// TwinCAT 3 PLC project TcOpcUaServer_Testproject
// ProgramVersion: 3.1.4022.3
// libraries:
//   Tc2_MPBus, * (Beckhoff Automation GmbH)
//   Tc2_Standard, * (Beckhoff Automation GmbH)
//   Tc2_System, * (Beckhoff Automation GmbH)
//   Tc3_Interfaces, * (Beckhoff Automation GmbH)
//   Tc3_Module, * (Beckhoff Automation GmbH)
// project tree:
//   DUTs/Enums/ E_Enum_2.TcDUT, E_Operation.TcDUT, E_Enum_1.TcDUT (not stored)
//   DUTs/Structures/ ST_Complex_1.TcDUT, ST_Complex_3.TcDUT, ST_Complex_4.TcDUT, ST_Complex_5.TcDUT (not stored), ST_Complex_6.TcDUT, ST_Complex_7.TcDUT, ST_Complex_8.TcDUT, ST_MathematicResults.TcDUT (not stored), ST_MathOperation.TcDUT, ST_Complex_2.TcDUT (not stored)
//   GVLs/ GVL_alarm_condition.TcGVL (not stored), GVL_analog_items.TcGVL, GVL_historizing.TcGVL (not stored), GVL_inheritance.TcGVL (not stored), GVL_user_access.TcGVL, Settings.TcGVL (not stored), GVL_arrays.TcGVL, GVL_enums.TcGVL, GVL_methods.TcGVL (not stored), GVL_structures.TcGVL (not stored), GVL_nodes_dynamic.TcGVL, GVL_nodes_static.TcGVL
//   / PlcTask.TcTTO (not stored)
//   POUs/Inheritance/ FB_Base.TcPOU (not stored), FB_Derived.TcPOU (not stored)
//   POUs/ MAIN.TcPOU (not stored)
//   POUs/Methods/ FB_Mathematics.TcPOU (not stored), FB_Methods.TcPOU
//   POUs/Programs/ PRG_Dynamic.TcPOU, PRG_Static.TcPOU
// real-time tasks:
//   TASK PlcTask: cycle T#10ms, priority 20, ADS port 350

// ---- DUTs/Enums/E_Enum_2.TcDUT
TYPE E_Enum_2 :
(
	ZERO := 0,
	ONE := 1,
	TWO := 2,
	THREE := 3,
	THIRTEEN := 13,
	the_answer_to_life_the_universe_and_everything := 42
) INT;
END_TYPE

// ---- DUTs/Enums/E_Operation.TcDUT
TYPE E_Operation :
(
	Addition := 0,
	Substract,
	Multiply,
	Divide
);
END_TYPE

// ---- DUTs/Structures/ST_Complex_1.TcDUT
{attribute 'OPC.UA.DA' := '1'}
{attribute 'OPC.UA.DA.StructuredType' := '1'}
TYPE ST_Complex_1 :
STRUCT
	x 	: E_Enum_1;
	a 	: DINT;
	str : STRING;
	b 	: DINT;
END_STRUCT
END_TYPE

// ---- DUTs/Structures/ST_Complex_3.TcDUT
{attribute 'OPC.UA.DA' := '1'}
{attribute 'OPC.UA.DA.StructuredType' := '1'}
TYPE ST_Complex_3 :
STRUCT
	ErrorID : MP_ERROR;
END_STRUCT
END_TYPE

// ---- DUTs/Structures/ST_Complex_4.TcDUT
{attribute 'OPC.UA.DA' := '1'}
{attribute 'OPC.UA.DA.StructuredType' := '1'}
TYPE ST_Complex_4 :
STRUCT
	ErrorID : E_Enum_1;
END_STRUCT
END_TYPE

// ---- DUTs/Structures/ST_Complex_6.TcDUT
TYPE ST_Complex_6 :
STRUCT
	a : INT := 42;
	b : DINT := 43;
	c : REAL := 42.42;
	d : LREAL := 42.42;
	e : INT := 44;
	f : BOOL := TRUE;
END_STRUCT
END_TYPE

// ---- DUTs/Structures/ST_Complex_7.TcDUT
TYPE ST_Complex_7 :
STRUCT
	a : LREAL := 42.42;
	b : REAL := 42.42;
	c : REAL := 42.42;
END_STRUCT
END_TYPE

// ---- DUTs/Structures/ST_Complex_8.TcDUT
{attribute 'OPC.UA.DA' := '1'}
{attribute 'OPC.UA.DA.StructuredType' := '1'}
TYPE ST_Complex_8 :
STRUCT
	stComplex		: ST_Complex_1;
	strString5		: STRING[5]; (*String, max 5 chars*)
	eEnum	 		: E_Enum_1;
	strString3	 	: STRING[3]; (*String, max 3 chars*)
	arrComplex 		: ARRAY[0..1] OF ST_Complex_1;
	arrDint		 	: ARRAY[0..100] OF DINT;	
END_STRUCT
END_TYPE

// ---- DUTs/Structures/ST_MathOperation.TcDUT
{attribute 'OPC.UA.DA.Description' := 'Structure to describe a math operation having one operator and two oparands'}
TYPE ST_MathOperation :
STRUCT
	operator : E_OPERATION; (*define the operator for calculation*)
	a : LREAL; (*First operand*)
	b : LREAL; (*Second operand*)
END_STRUCT
END_TYPE

// ---- GVLs/GVL_analog_items.TcGVL
{attribute 'qualified_only'}
VAR_GLOBAL
	{attribute 'OPC.UA.DA' := '1'}
	{attribute 'OPC.UA.DA.AnalogItemType' := '1'}
	{attribute 'OPC.UA.DA.AnalogItemType.EngineeringUnits' := '20529'  }(*EngeneeringUnit = percent*)
	{attribute 'OPC.UA.DA.AnalogItemType.InstrumentRange' := '0:100'  }
	{attribute 'OPC.UA.DA.AnalogItemType.EURange' := '10:90'  }
	{attribute 'OPC.UA.DA.AnalogItemType.WriteBehavior' := '1'  } (*AnalogWrMode_AllowAny = 0,
																	AnalogWrMode_Clamp = 1,
																	AnalogWrMode_Reject = 2,*)
	{attribute 'OPC.UA.DA.Description' := 'Analog item type. Write mode is clamped to instrument range'}
	analog_percent : REAL := 50;
	
	{attribute 'OPC.UA.DA' := '1'}
	{attribute 'OPC.UA.DA.AnalogItemType' := '1'}
	{attribute 'OPC.UA.DA.AnalogItemType.EngineeringUnits' := '12851'  }(*EngeneeringUnit = gram_per_cubic_centimetre*)
	{attribute 'OPC.UA.DA.AnalogItemType.InstrumentRange' := '0:100'  }
	{attribute 'OPC.UA.DA.AnalogItemType.EURange' := '0:75'  }
	{attribute 'OPC.UA.DA.AnalogItemType.WriteBehavior' := '2'  } (*AnalogWrMode_AllowAny = 0,
																	AnalogWrMode_Clamp = 1,
																	AnalogWrMode_Reject = 2,*)
	{attribute 'OPC.UA.DA.Description' := 'Analog item type. Write is rejected when out of instrument range'}
	analog_gram_per_cubic_centimetre : REAL := 50;	
	
	{attribute 'OPC.UA.DA' := '1'}
	{attribute 'OPC.UA.DA.AnalogItemType' := '1'}
	{attribute 'OPC.UA.DA.AnalogItemType.EngineeringUnits' := '5257525'  }(*EngeneeringUnit = megabyte_per_second*)
	{attribute 'OPC.UA.DA.AnalogItemType.EURange' := '0:10'  }
	{attribute 'OPC.UA.DA.AnalogItemType.InstrumentRange' := '0:100'  }
	{attribute 'OPC.UA.DA.AnalogItemType.WriteBehavior' := '0'  } (*AnalogWrMode_AllowAny = 0,
																	AnalogWrMode_Clamp = 1,
																	AnalogWrMode_Reject = 2,*)
	{attribute 'OPC.UA.DA.Description' := 'Analog item type. Write mode allows writing out of Instrument range'}
	analog_mbps : REAL;	
	
	{attribute 'OPC.UA.DA' := '1'}
	{attribute 'OPC.UA.DA.AnalogItemType' := '1'}
	{attribute 'OPC.UA.DA.AnalogItemType.EngineeringUnits' := '20529'  }(*EngeneeringUnit = percent*)
	{attribute 'OPC.UA.DA.AnalogItemType.InstrumentRange' := '0:100'  }
	{attribute 'OPC.UA.DA.AnalogItemType.EURange' := '10:90'  }
	{attribute 'OPC.UA.DA.AnalogItemType.WriteBehavior' := '2'  } (*AnalogWrMode_AllowAny = 0,
																	AnalogWrMode_Clamp = 1,
																	AnalogWrMode_Reject = 2,*)
	{attribute 'OPC.UA.DA.Description' := 'Analog item of type Double. '}
	analog_dbl : LREAL := 50;	
	
	{attribute 'OPC.UA.DA' := '1'}
	{attribute 'OPC.UA.DA.AnalogItemType' := '1'}
	{attribute 'OPC.UA.DA.AnalogItemType.EngineeringUnits' := '20529'  }(*EngeneeringUnit = percent*)
	{attribute 'OPC.UA.DA.AnalogItemType.InstrumentRange' := '0:100'  }
	{attribute 'OPC.UA.DA.AnalogItemType.EURange' := '10:90'  }
	{attribute 'OPC.UA.DA.AnalogItemType.WriteBehavior' := '2'  } (*AnalogWrMode_AllowAny = 0,
																	AnalogWrMode_Clamp = 1,
																	AnalogWrMode_Reject = 2,*)
	{attribute 'OPC.UA.DA.Description' := 'Analog item of type Float. '}
	analog_flt : REAL := 50;		
	
	{attribute 'OPC.UA.DA' := '1'}
	{attribute 'OPC.UA.DA.AnalogItemType' := '1'}
	{attribute 'OPC.UA.DA.AnalogItemType.EngineeringUnits' := '20529'  }(*EngeneeringUnit = percent*)
	{attribute 'OPC.UA.DA.AnalogItemType.InstrumentRange' := '0:100'  }
	{attribute 'OPC.UA.DA.AnalogItemType.EURange' := '10:90'  }
	{attribute 'OPC.UA.DA.AnalogItemType.WriteBehavior' := '2'  } (*AnalogWrMode_AllowAny = 0,
																	AnalogWrMode_Clamp = 1,
																	AnalogWrMode_Reject = 2,*)
	{attribute 'OPC.UA.DA.Description' := 'Analog item of type Int16. '}
	analog_i16 : INT := 50;		
	
	{attribute 'OPC.UA.DA' := '1'}
	{attribute 'OPC.UA.DA.AnalogItemType' := '1'}
	{attribute 'OPC.UA.DA.AnalogItemType.EngineeringUnits' := '20529'  }(*EngeneeringUnit = percent*)
	{attribute 'OPC.UA.DA.AnalogItemType.InstrumentRange' := '0:100'  }
	{attribute 'OPC.UA.DA.AnalogItemType.EURange' := '10:90'  }
	{attribute 'OPC.UA.DA.AnalogItemType.WriteBehavior' := '2'  } (*AnalogWrMode_AllowAny = 0,
																	AnalogWrMode_Clamp = 1,
																	AnalogWrMode_Reject = 2,*)
	{attribute 'OPC.UA.DA.Description' := 'Analog item of type UInt16. '}
	analog_ui16 : UINT := 50;		
	
	{attribute 'OPC.UA.DA' := '1'}
	{attribute 'OPC.UA.DA.AnalogItemType' := '1'}
	{attribute 'OPC.UA.DA.AnalogItemType.EngineeringUnits' := '20529'  }(*EngeneeringUnit = percent*)
	{attribute 'OPC.UA.DA.AnalogItemType.InstrumentRange' := '0:100'  }
	{attribute 'OPC.UA.DA.AnalogItemType.EURange' := '10:90'  }
	{attribute 'OPC.UA.DA.AnalogItemType.WriteBehavior' := '2'  } (*AnalogWrMode_AllowAny = 0,
																	AnalogWrMode_Clamp = 1,
																	AnalogWrMode_Reject = 2,*)
	{attribute 'OPC.UA.DA.Description' := 'Analog item of type Int32. '}
	analog_i32 : DINT := 50;		

	{attribute 'OPC.UA.DA' := '1'}
	{attribute 'OPC.UA.DA.AnalogItemType' := '1'}
	{attribute 'OPC.UA.DA.AnalogItemType.EngineeringUnits' := '20529'  }(*EngeneeringUnit = percent*)
	{attribute 'OPC.UA.DA.AnalogItemType.InstrumentRange' := '0:100'  }
	{attribute 'OPC.UA.DA.AnalogItemType.EURange' := '10:90'  }
	{attribute 'OPC.UA.DA.AnalogItemType.WriteBehavior' := '2'  } (*AnalogWrMode_AllowAny = 0,
																	AnalogWrMode_Clamp = 1,
																	AnalogWrMode_Reject = 2,*)
	{attribute 'OPC.UA.DA.Description' := 'Analog item of type UInt32. '}
	analog_ui32 : UDINT := 50;
	
	{attribute 'OPC.UA.DA' := '1'}
	{attribute 'OPC.UA.DA.AnalogItemType' := '1'}
	{attribute 'OPC.UA.DA.AnalogItemType.EngineeringUnits' := '20529'  }(*EngeneeringUnit = percent*)
	{attribute 'OPC.UA.DA.AnalogItemType.InstrumentRange' := '0:100'  }
	{attribute 'OPC.UA.DA.AnalogItemType.EURange' := '10:90'  }
	{attribute 'OPC.UA.DA.AnalogItemType.WriteBehavior' := '2'  } (*AnalogWrMode_AllowAny = 0,
																	AnalogWrMode_Clamp = 1,
																	AnalogWrMode_Reject = 2,*)
	{attribute 'OPC.UA.DA.Description' := 'Analog item of type Int64. '}
	analog_i64 : LINT := 50;		
	
	{attribute 'OPC.UA.DA' := '1'}
	{attribute 'OPC.UA.DA.AnalogItemType' := '1'}
	{attribute 'OPC.UA.DA.AnalogItemType.EngineeringUnits' := '20529'  }(*EngeneeringUnit = percent*)
	{attribute 'OPC.UA.DA.AnalogItemType.InstrumentRange' := '0:100'  }
	{attribute 'OPC.UA.DA.AnalogItemType.EURange' := '10:90'  }
	{attribute 'OPC.UA.DA.AnalogItemType.WriteBehavior' := '2'  } (*AnalogWrMode_AllowAny = 0,
																	AnalogWrMode_Clamp = 1,
																	AnalogWrMode_Reject = 2,*)
	{attribute 'OPC.UA.DA.Description' := 'Analog item of type UInt64. '}
	analog_ui64 : ULINT := 50;		
	
	{attribute 'OPC.UA.DA' := '1'}
	{attribute 'OPC.UA.DA.AnalogItemType' := '1'}
	{attribute 'OPC.UA.DA.AnalogItemType.EngineeringUnits' := '20529'  }(*EngeneeringUnit = percent*)
	{attribute 'OPC.UA.DA.AnalogItemType.InstrumentRange' := '0:100'  }
	{attribute 'OPC.UA.DA.AnalogItemType.EURange' := '10:90'  }
	{attribute 'OPC.UA.DA.AnalogItemType.WriteBehavior' := '2'  } (*AnalogWrMode_AllowAny = 0,
																	AnalogWrMode_Clamp = 1,
																	AnalogWrMode_Reject = 2,*)
	{attribute 'OPC.UA.DA.Description' := 'Analog item of type SByte. '}
	analog_i8 : SINT := 50;		
	
	{attribute 'OPC.UA.DA' := '1'}
	{attribute 'OPC.UA.DA.AnalogItemType' := '1'}
	{attribute 'OPC.UA.DA.AnalogItemType.EngineeringUnits' := '20529'  }(*EngeneeringUnit = percent*)
	{attribute 'OPC.UA.DA.AnalogItemType.InstrumentRange' := '0:100'  }
	{attribute 'OPC.UA.DA.AnalogItemType.EURange' := '10:90'  }
	{attribute 'OPC.UA.DA.AnalogItemType.WriteBehavior' := '2'  } (*AnalogWrMode_AllowAny = 0,
																	AnalogWrMode_Clamp = 1,
																	AnalogWrMode_Reject = 2,*)
	{attribute 'OPC.UA.DA.Description' := 'Analog item of type Byte. '}
	analog_ui8 : USINT := 50;	
END_VAR

// ---- GVLs/GVL_user_access.TcGVL
{attribute 'qualified_only'}
VAR_GLOBAL
	{attribute 'OPC.UA.DA' := '1'}
	{attribute 'OPC.UA.DA.Description' := 'read only for user1'}	
	user1_R		: INT;
	{attribute 'OPC.UA.DA' := '1'}
	{attribute 'OPC.UA.DA.Description' := 'read writeable for user1'}	
	user1_RW	: INT;
	{attribute 'OPC.UA.DA' := '1'}
	{attribute 'OPC.UA.DA.Description' := 'write only for user1'}	
	user1_W	: INT;
	{attribute 'OPC.UA.DA' := '1'}
	{attribute 'OPC.UA.DA.Description' := 'read only for user1'}	
	user2_R		: INT;
	{attribute 'OPC.UA.DA' := '1'}
	{attribute 'OPC.UA.DA.Description' := 'read writeable for user1'}	
	user2_RW	: INT;
	{attribute 'OPC.UA.DA' := '1'}
	{attribute 'OPC.UA.DA.Description' := 'write only for user1'}	
	user2_W	: INT;	
	{attribute 'OPC.UA.DA' := '1'}
	{attribute 'OPC.UA.DA.Description' := 'read/ writeable for user1, read only for user 2'}	
	user1_RW_user2_R	: INT;
END_VAR

// ---- GVLs/GVL_arrays.TcGVL
{attribute 'qualified_only'}
VAR_GLOBAL
	{attribute 'OPC.UA.DA' := '1'}
	{attribute 'OPC.UA.DA.StructuredType' := '1'}
	{attribute 'OPC.UA.DA.Description' := 'Complex (structured) type'} 	
	arrStComplex : ARRAY[0..ARRSIZEX] OF ST_Complex_1;

	{attribute 'OPC.UA.DA' := '1'}
	{attribute 'OPC.UA.DA.StructuredType' := '1'}
	{attribute 'OPC.UA.DA.Description' := 'Complex (structured) type'} 		
	arrStComplex2 : ARRAY[0..ARRSIZEX] OF ST_Complex_2;	
END_VAR

// ---- GVLs/GVL_enums.TcGVL
{attribute 'qualified_only'}
VAR_GLOBAL
	{attribute 'OPC.UA.DA' := '1'}
	{attribute 'OPC.UA.DA.Description' := 'Enumeration type (DINT)'} 
	Enum1 : E_Enum_1;
	{attribute 'OPC.UA.DA' := '1'}
	{attribute 'OPC.UA.DA.Description' := 'Enumeration type (INT)'} 
	Enum2 : E_Enum_2;	
END_VAR

// ---- GVLs/GVL_nodes_dynamic.TcGVL
VAR_GLOBAL
	//scalars
	{attribute 'OPC.UA.DA' := '1'}
	{attribute 'OPC.UA.DA.Description' := 'Scalar BOOL'} 
	dyn_scalar_BOOL	: BOOL;(* ~ 	(OPC : 1 : available for OPC-clients) *)
	{attribute 'OPC.UA.DA' := '1'}
	{attribute 'OPC.UA.DA.Description' := 'Scalar SINT'}
	dyn_scalar_I1	: SINT;		(* ~ 	(OPC : 1 : available for OPC-clients) *)					
	{attribute 'OPC.UA.DA' := '1'}
	{attribute 'OPC.UA.DA.Description' := 'Scalar USINT'}	
	dyn_scalar_UI1	: USINT;	(* ~ 	(OPC : 1 : available for OPC-clients) *)					
	{attribute 'OPC.UA.DA' := '1'}
	{attribute 'OPC.UA.DA.Description' := 'Scalar INT'}	
	dyn_scalar_I2 	: INT;			(* ~ 	(OPC : 1 : available for OPC-clients) *)				
	{attribute 'OPC.UA.DA' := '1'}
	{attribute 'OPC.UA.DA.Description' := 'Scalar UINT'}	
	dyn_scalar_UI2	: UINT;			(* ~ 	(OPC : 1 : available for OPC-clients) *)				
	{attribute 'OPC.UA.DA' := '1'}
	{attribute 'OPC.UA.DA.Description' := 'Scalar DINT'}	
	dyn_scalar_I4	: DINT;		(* ~ 	(OPC : 1 : available for OPC-clients) *)					
	{attribute 'OPC.UA.DA' := '1'}
	{attribute 'OPC.UA.DA.Description' := 'Scalar UDINT'}	
	dyn_scalar_UI4	: UDINT;(* ~ 	(OPC : 1 : available for OPC-clients) *)
	{attribute 'OPC.UA.DA' := '1'}
	{attribute 'OPC.UA.DA.Description' := 'Scalar LINT'}
	dyn_scalar_I8	: LINT;	(* ~ 	(OPC : 1 : available for OPC-clients) *)
	{attribute 'OPC.UA.DA' := '1'}
	{attribute 'OPC.UA.DA.Description' := 'Scalar ULINT'}
	dyn_scalar_UI8	: ULINT;(* ~ 	(OPC : 1 : available for OPC-clients) *)
	{attribute 'OPC.UA.DA' := '1'}
	{attribute 'OPC.UA.DA.Description' := 'Scalar BYTE'}
	dyn_scalar_BYTE	: BYTE;(* ~ 	(OPC : 1 : available for OPC-clients) *)
	{attribute 'OPC.UA.DA' := '1'}
	{attribute 'OPC.UA.DA.Description' := 'Scalar WORD'}	
	dyn_scalar_WORD	: WORD;(* ~ 	(OPC : 1 : available for OPC-clients) *)
	{attribute 'OPC.UA.DA' := '1'}
	{attribute 'OPC.UA.DA.Description' := 'Scalar DWORD'}	
	dyn_scalar_DWORD: DWORD;(* ~ 	(OPC : 1 : available for OPC-clients) *)
	{attribute 'OPC.UA.DA' := '1'}
	{attribute 'OPC.UA.DA.Description' := 'Scalar LWORD'}	
	dyn_scalar_LWORD: LWORD;(* ~ 	(OPC : 1 : available for OPC-clients) *)
	{attribute 'OPC.UA.DA' := '1'}
	{attribute 'OPC.UA.DA.Description' := 'Scalar REAL'}	
	dyn_scalar_R4	: REAL;(* ~ 	(OPC : 1 : available for OPC-clients) *)
	{attribute 'OPC.UA.DA' := '1'}
	{attribute 'OPC.UA.DA.Description' := 'Scalar LREAL'}
	dyn_scalar_R8	: LREAL;(* ~ 	(OPC : 1 : available for OPC-clients) *)
	{attribute 'OPC.UA.DA' := '1'}
	{attribute 'OPC.UA.DA.Description' := 'Scalar STRING'}	
	dyn_scalar_BSTR	: STRING;(* ~ 	(OPC : 1 : available for OPC-clients) *)
	{attribute 'OPC.UA.DA' := '1'}
	{attribute 'OPC.UA.DA.Description' := 'Scalar CHAR'}	
	//dyn_scalar_CHAR	: CHAR;
	{attribute 'OPC.UA.DA' := '1'}
	{attribute 'OPC.UA.DA.Description' := 'Scalar WSTRING'}	
	dyn_scalar_WSTRING : WSTRING;(* ~ 	(OPC : 1 : available for OPC-clients) *)
	{attribute 'OPC.UA.DA' := '1'}
	{attribute 'OPC.UA.DA.Description' := 'Scalar WCHAR'}	
	//dyn_scalar_WCHAR: WCHAR;
	{attribute 'OPC.UA.DA' := '1'}
	{attribute 'OPC.UA.DA.Description' := 'Scalar DT'}	
	dyn_scalar_DT	: DT;(* ~ 	(OPC : 1 : available for OPC-clients) *)
	{attribute 'OPC.UA.DA' := '1'}
	{attribute 'OPC.UA.DA.Description' := 'Scalar DATE'}	
	dyn_scalar_DATE : DATE;(* ~ 	(OPC : 1 : available for OPC-clients) *)
	{attribute 'OPC.UA.DA' := '1'}
	{attribute 'OPC.UA.DA.Description' := 'Scalar TOD'}	
	dyn_scalar_TOD	: TOD;(* ~ 	(OPC : 1 : available for OPC-clients) *)
	{attribute 'OPC.UA.DA' := '1'}
	{attribute 'OPC.UA.DA.Description' := 'Scalar TIME'}	
	dyn_scalar_TIME	: TIME;(* ~ 	(OPC : 1 : available for OPC-clients) *)
	
	//1dim
	{attribute 'OPC.UA.DA' := '1'}
	{attribute 'OPC.UA.DA.Description' := '1dim Array BOOL'}	
	dyn_1dim_BOOL	: ARRAY[0..ARRSIZEX] OF BOOL;(* ~ 	(OPC : 1 : available for OPC-clients) *)
	{attribute 'OPC.UA.DA' := '1'}
	{attribute 'OPC.UA.DA.Description' := '1dim Array BOOL'}	
	dyn_1dim_I1		: ARRAY[0..ARRSIZEX] OF SINT;(* ~ 	(OPC : 1 : available for OPC-clients) *)
	{attribute 'OPC.UA.DA' := '1'}
	{attribute 'OPC.UA.DA.Description' := '1dim Array BOOL'}	
	dyn_1dim_I1_Huge: ARRAY[0..ARRSIZEHUGE] OF SINT;(* ~ 	(OPC : 1 : available for OPC-clients) *)	
	{attribute 'OPC.UA.DA' := '1'}
	{attribute 'OPC.UA.DA.Description' := '1dim Array BOOL'}
	dyn_1dim_UI1	: ARRAY[0..ARRSIZEX] OF USINT;(* ~ 	(OPC : 1 : available for OPC-clients) *)
	{attribute 'OPC.UA.DA' := '1'}
	{attribute 'OPC.UA.DA.Description' := '1dim Array BOOL'}
	dyn_1dim_I2 	: ARRAY[0..ARRSIZEX] OF INT;(* ~ 	(OPC : 1 : available for OPC-clients) *)
	{attribute 'OPC.UA.DA' := '1'}
	{attribute 'OPC.UA.DA.Description' := '1dim Array BOOL'}	
	dyn_1dim_UI2	: ARRAY[0..ARRSIZEX] OF UINT;(* ~ 	(OPC : 1 : available for OPC-clients) *)
	{attribute 'OPC.UA.DA' := '1'}
	{attribute 'OPC.UA.DA.Description' := '1dim Array BOOL'}	
	dyn_1dim_I4		: ARRAY[0..ARRSIZEX] OF DINT;(* ~ 	(OPC : 1 : available for OPC-clients) *)
	{attribute 'OPC.UA.DA' := '1'}
	{attribute 'OPC.UA.DA.Description' := '1dim Array BOOL'}	
	dyn_1dim_I4_Huge: ARRAY[0..ARRSIZEHUGE] OF DINT;(* ~ 	(OPC : 1 : available for OPC-clients) *)	
	{attribute 'OPC.UA.DA' := '1'}
	{attribute 'OPC.UA.DA.Description' := '1dim Array BOOL'}
	dyn_1dim_UI4	: ARRAY[0..ARRSIZEX] OF UDINT;(* ~ 	(OPC : 1 : available for OPC-clients) *)
	{attribute 'OPC.UA.DA' := '1'}
	{attribute 'OPC.UA.DA.Description' := '1dim Array BOOL'}
	dyn_1dim_I8		: ARRAY[0..ARRSIZEX] OF LINT;(* ~ 	(OPC : 1 : available for OPC-clients) *)
	{attribute 'OPC.UA.DA' := '1'}
	{attribute 'OPC.UA.DA.Description' := '1dim Array BOOL'}
	dyn_1dim_UI8	: ARRAY[0..ARRSIZEX] OF ULINT;(* ~ 	(OPC : 1 : available for OPC-clients) *)
	{attribute 'OPC.UA.DA' := '1'}
	{attribute 'OPC.UA.DA.Description' := '1dim Array BOOL'}
	dyn_1dim_BYTE	: ARRAY[0..ARRSIZEX] OF BYTE;(* ~ 	(OPC : 1 : available for OPC-clients) *)
	{attribute 'OPC.UA.DA' := '1'}
	{attribute 'OPC.UA.DA.Description' := '1dim Array BOOL'}
	dyn_1dim_WORD	: ARRAY[0..ARRSIZEX] OF WORD;(* ~ 	(OPC : 1 : available for OPC-clients) *)
	{attribute 'OPC.UA.DA' := '1'}
	{attribute 'OPC.UA.DA.Description' := '1dim Array BOOL'}
	dyn_1dim_DWORD	: ARRAY[0..ARRSIZEX] OF DWORD;(* ~ 	(OPC : 1 : available for OPC-clients) *)
	{attribute 'OPC.UA.DA' := '1'}
	{attribute 'OPC.UA.DA.Description' := '1dim Array BOOL'}
	dyn_1dim_LWORD	: ARRAY[0..ARRSIZEX] OF LWORD;(* ~ 	(OPC : 1 : available for OPC-clients) *)
	{attribute 'OPC.UA.DA' := '1'}
	{attribute 'OPC.UA.DA.Description' := '1dim Array BOOL'}
	dyn_1dim_R4		: ARRAY[0..ARRSIZEX] OF REAL;(* ~ 	(OPC : 1 : available for OPC-clients) *)
	{attribute 'OPC.UA.DA' := '1'}
	{attribute 'OPC.UA.DA.Description' := '1dim Array BOOL'}
	dyn_1dim_R8		: ARRAY[0..ARRSIZEX] OF LREAL;(* ~ 	(OPC : 1 : available for OPC-clients) *)
	{attribute 'OPC.UA.DA' := '1'}
	{attribute 'OPC.UA.DA.Description' := '1dim Array BOOL'}
	dyn_1dim_BSTR	: ARRAY[0..ARRSIZEX] OF STRING;(* ~ 	(OPC : 1 : available for OPC-clients) *)
	{attribute 'OPC.UA.DA' := '1'}
	{attribute 'OPC.UA.DA.Description' := '1dim Array BOOL'}
	//dyn_1dim_CHAR	: ARRAY[0..ARRSIZEX] OF CHAR;
	{attribute 'OPC.UA.DA' := '1'}
	{attribute 'OPC.UA.DA.Description' := '1dim Array BOOL'}
	dyn_1dim_WSTRING : ARRAY[0..ARRSIZEX] OF WSTRING;(* ~ 	(OPC : 1 : available for OPC-clients) *)
	{attribute 'OPC.UA.DA' := '1'}
	{attribute 'OPC.UA.DA.Description' := '1dim Array BOOL'}
	//dyn_1dim_WCHAR: ARRAY[0..ARRSIZEX] OF WCHAR;
	{attribute 'OPC.UA.DA' := '1'}
	{attribute 'OPC.UA.DA.Description' := '1dim Array BOOL'}
	dyn_1dim_DT		: ARRAY[0..ARRSIZEX] OF DT;(* ~ 	(OPC : 1 : available for OPC-clients) *)
	{attribute 'OPC.UA.DA' := '1'}
	{attribute 'OPC.UA.DA.Description' := '1dim Array BOOL'}
	dyn_1dim_DATE 	: ARRAY[0..ARRSIZEX] OF DATE;(* ~ 	(OPC : 1 : available for OPC-clients) *)
	{attribute 'OPC.UA.DA' := '1'}
	{attribute 'OPC.UA.DA.Description' := '1dim Array BOOL'}
	dyn_1dim_TOD	: ARRAY[0..ARRSIZEX] OF TOD;(* ~ 	(OPC : 1 : available for OPC-clients) *)
	{attribute 'OPC.UA.DA' := '1'}
	{attribute 'OPC.UA.DA.Description' := '1dim Array BOOL'}
	dyn_1dim_TIME	: ARRAY[0..ARRSIZEX] OF TIME;(* ~ 	(OPC : 1 : available for OPC-clients) *)
	
	//2dim
	{attribute 'OPC.UA.DA' := '1'}
	{attribute 'OPC.UA.DA.Description' := '2dim Array BOOL'}
	dyn_2dim_BOOL	: ARRAY[0..ARRSIZEX, 0..ARRSIZEY] OF BOOL;(* ~ 	(OPC : 1 : available for OPC-clients) *)
	{attribute 'OPC.UA.DA' := '1'}
	{attribute 'OPC.UA.DA.Description' := '2dim Array BOOL'}
	dyn_2dim_I1		: ARRAY[0..ARRSIZEX, 0..ARRSIZEY] OF SINT;(* ~ 	(OPC : 1 : available for OPC-clients) *)
	{attribute 'OPC.UA.DA' := '1'}
	{attribute 'OPC.UA.DA.Description' := '2dim Array BOOL'}
	dyn_2dim_UI1	: ARRAY[0..ARRSIZEX, 0..ARRSIZEY] OF USINT;(* ~ 	(OPC : 1 : available for OPC-clients) *)
	{attribute 'OPC.UA.DA' := '1'}
	{attribute 'OPC.UA.DA.Description' := '2dim Array BOOL'}
	dyn_2dim_I2 	: ARRAY[0..ARRSIZEX, 0..ARRSIZEY] OF INT;(* ~ 	(OPC : 1 : available for OPC-clients) *)
	{attribute 'OPC.UA.DA' := '1'}
	{attribute 'OPC.UA.DA.Description' := '2dim Array BOOL'}
	dyn_2dim_UI2	: ARRAY[0..ARRSIZEX, 0..ARRSIZEY] OF UINT;(* ~ 	(OPC : 1 : available for OPC-clients) *)
	{attribute 'OPC.UA.DA' := '1'}
	{attribute 'OPC.UA.DA.Description' := '2dim Array BOOL'}
	dyn_2dim_I4		: ARRAY[0..ARRSIZEX, 0..ARRSIZEY] OF DINT;(* ~ 	(OPC : 1 : available for OPC-clients) *)
	{attribute 'OPC.UA.DA' := '1'}
	{attribute 'OPC.UA.DA.Description' := '2dim Array BOOL'}
	dyn_2dim_UI4	: ARRAY[0..ARRSIZEX, 0..ARRSIZEY] OF UDINT;(* ~ 	(OPC : 1 : available for OPC-clients) *)
	{attribute 'OPC.UA.DA' := '1'}
	{attribute 'OPC.UA.DA.Description' := '2dim Array BOOL'}
	dyn_2dim_I8		: ARRAY[0..ARRSIZEX, 0..ARRSIZEY] OF LINT;(* ~ 	(OPC : 1 : available for OPC-clients) *)
	{attribute 'OPC.UA.DA' := '1'}
	{attribute 'OPC.UA.DA.Description' := '2dim Array BOOL'}
	dyn_2dim_UI8	: ARRAY[0..ARRSIZEX, 0..ARRSIZEY] OF ULINT;(* ~ 	(OPC : 1 : available for OPC-clients) *)
	{attribute 'OPC.UA.DA' := '1'}
	{attribute 'OPC.UA.DA.Description' := '2dim Array BOOL'}
	dyn_2dim_BYTE	: ARRAY[0..ARRSIZEX, 0..ARRSIZEY] OF BYTE;(* ~ 	(OPC : 1 : available for OPC-clients) *)
	{attribute 'OPC.UA.DA' := '1'}
	{attribute 'OPC.UA.DA.Description' := '2dim Array BOOL'}
	dyn_2dim_WORD	: ARRAY[0..ARRSIZEX, 0..ARRSIZEY] OF WORD;(* ~ 	(OPC : 1 : available for OPC-clients) *)
	{attribute 'OPC.UA.DA' := '1'}
	{attribute 'OPC.UA.DA.Description' := '2dim Array BOOL'}
	dyn_2dim_DWORD	: ARRAY[0..ARRSIZEX, 0..ARRSIZEY] OF DWORD;(* ~ 	(OPC : 1 : available for OPC-clients) *)
	{attribute 'OPC.UA.DA' := '1'}
	{attribute 'OPC.UA.DA.Description' := '2dim Array BOOL'}
	dyn_2dim_LWORD	: ARRAY[0..ARRSIZEX, 0..ARRSIZEY] OF LWORD;(* ~ 	(OPC : 1 : available for OPC-clients) *)
	{attribute 'OPC.UA.DA' := '1'}
	{attribute 'OPC.UA.DA.Description' := '2dim Array BOOL'}
	dyn_2dim_R4		: ARRAY[0..ARRSIZEX, 0..ARRSIZEY] OF REAL;(* ~ 	(OPC : 1 : available for OPC-clients) *)
	{attribute 'OPC.UA.DA' := '1'}
	{attribute 'OPC.UA.DA.Description' := '2dim Array BOOL'}
	dyn_2dim_R8		: ARRAY[0..ARRSIZEX, 0..ARRSIZEY] OF LREAL;(* ~ 	(OPC : 1 : available for OPC-clients) *)
	{attribute 'OPC.UA.DA' := '1'}
	{attribute 'OPC.UA.DA.Description' := '2dim Array BOOL'}
	dyn_2dim_BSTR	: ARRAY[0..ARRSIZEX, 0..ARRSIZEY] OF STRING;(* ~ 	(OPC : 1 : available for OPC-clients) *)
	{attribute 'OPC.UA.DA' := '1'}
	{attribute 'OPC.UA.DA.Description' := '2dim Array BOOL'}
	//dyn_2dim_CHAR	: ARRAY[0..ARRSIZEX, 0..ARRSIZEY] OF CHAR;
	{attribute 'OPC.UA.DA' := '1'}
	{attribute 'OPC.UA.DA.Description' := '2dim Array BOOL'}
	dyn_2dim_WSTRING : ARRAY[0..ARRSIZEX, 0..ARRSIZEY] OF WSTRING;(* ~ 	(OPC : 1 : available for OPC-clients) *)
	{attribute 'OPC.UA.DA' := '1'}
	{attribute 'OPC.UA.DA.Description' := '2dim Array BOOL'}
	//dyn_2dim_WCHAR: ARRAY[0..ARRSIZEX, 0..ARRSIZEY] OF WCHAR;
	{attribute 'OPC.UA.DA' := '1'}
	{attribute 'OPC.UA.DA.Description' := '2dim Array BOOL'}
	dyn_2dim_DT		: ARRAY[0..ARRSIZEX, 0..ARRSIZEY] OF DT;(* ~ 	(OPC : 1 : available for OPC-clients) *)
	{attribute 'OPC.UA.DA' := '1'}
	{attribute 'OPC.UA.DA.Description' := '2dim Array BOOL'}
	dyn_2dim_DATE 	: ARRAY[0..ARRSIZEX, 0..ARRSIZEY] OF DATE;(* ~ 	(OPC : 1 : available for OPC-clients) *)
	{attribute 'OPC.UA.DA' := '1'}
	{attribute 'OPC.UA.DA.Description' := '2dim Array BOOL'}
	dyn_2dim_TOD	: ARRAY[0..ARRSIZEX, 0..ARRSIZEY] OF TOD;(* ~ 	(OPC : 1 : available for OPC-clients) *)
	{attribute 'OPC.UA.DA' := '1'}
	{attribute 'OPC.UA.DA.Description' := '2dim Array BOOL'}
	dyn_2dim_TIME	: ARRAY[0..ARRSIZEX, 0..ARRSIZEY] OF TIME;(* ~ 	(OPC : 1 : available for OPC-clients) *)

	//3dim
	{attribute 'OPC.UA.DA' := '1'}
	{attribute 'OPC.UA.DA.Description' := '3dim Array BOOL'}
	dyn_3dim_BOOL	: ARRAY[0..ARRSIZEX, 0..ARRSIZEY, 0..ARRSIZEZ] OF BOOL;(* ~ 	(OPC : 1 : available for OPC-clients) *)
	{attribute 'OPC.UA.DA' := '1'}
	{attribute 'OPC.UA.DA.Description' := '3dim Array BOOL'}
	dyn_3dim_I1		: ARRAY[0..ARRSIZEX, 0..ARRSIZEY, 0..ARRSIZEZ] OF SINT;(* ~ 	(OPC : 1 : available for OPC-clients) *)
	{attribute 'OPC.UA.DA' := '1'}
	{attribute 'OPC.UA.DA.Description' := '3dim Array BOOL'}
	dyn_3dim_UI1	: ARRAY[0..ARRSIZEX, 0..ARRSIZEY, 0..ARRSIZEZ] OF USINT;(* ~ 	(OPC : 1 : available for OPC-clients) *)
	{attribute 'OPC.UA.DA' := '1'}
	{attribute 'OPC.UA.DA.Description' := '3dim Array BOOL'}
	dyn_3dim_I2 	: ARRAY[0..ARRSIZEX, 0..ARRSIZEY, 0..ARRSIZEZ] OF INT;(* ~ 	(OPC : 1 : available for OPC-clients) *)
	{attribute 'OPC.UA.DA' := '1'}
	{attribute 'OPC.UA.DA.Description' := '3dim Array BOOL'}
	dyn_3dim_UI2	: ARRAY[0..ARRSIZEX, 0..ARRSIZEY, 0..ARRSIZEZ] OF UINT;(* ~ 	(OPC : 1 : available for OPC-clients) *)
	{attribute 'OPC.UA.DA' := '1'}
	{attribute 'OPC.UA.DA.Description' := '3dim Array BOOL'}
	dyn_3dim_I4		: ARRAY[0..ARRSIZEX, 0..ARRSIZEY, 0..ARRSIZEZ] OF DINT;(* ~ 	(OPC : 1 : available for OPC-clients) *)
	{attribute 'OPC.UA.DA' := '1'}
	{attribute 'OPC.UA.DA.Description' := '3dim Array BOOL'}
	dyn_3dim_UI4	: ARRAY[0..ARRSIZEX, 0..ARRSIZEY, 0..ARRSIZEZ] OF UDINT;(* ~ 	(OPC : 1 : available for OPC-clients) *)
	{attribute 'OPC.UA.DA' := '1'}
	{attribute 'OPC.UA.DA.Description' := '3dim Array BOOL'}
	dyn_3dim_I8		: ARRAY[0..ARRSIZEX, 0..ARRSIZEY, 0..ARRSIZEZ] OF LINT;(* ~ 	(OPC : 1 : available for OPC-clients) *)
	{attribute 'OPC.UA.DA' := '1'}
	{attribute 'OPC.UA.DA.Description' := '3dim Array BOOL'}
	dyn_3dim_UI8	: ARRAY[0..ARRSIZEX, 0..ARRSIZEY, 0..ARRSIZEZ] OF ULINT;(* ~ 	(OPC : 1 : available for OPC-clients) *)
	{attribute 'OPC.UA.DA' := '1'}
	{attribute 'OPC.UA.DA.Description' := '3dim Array BOOL'}
	dyn_3dim_BYTE	: ARRAY[0..ARRSIZEX, 0..ARRSIZEY, 0..ARRSIZEZ] OF BYTE;(* ~ 	(OPC : 1 : available for OPC-clients) *)
	{attribute 'OPC.UA.DA' := '1'}
	{attribute 'OPC.UA.DA.Description' := '3dim Array BOOL'}
	dyn_3dim_WORD	: ARRAY[0..ARRSIZEX, 0..ARRSIZEY, 0..ARRSIZEZ] OF WORD;(* ~ 	(OPC : 1 : available for OPC-clients) *)
	{attribute 'OPC.UA.DA' := '1'}
	{attribute 'OPC.UA.DA.Description' := '3dim Array BOOL'}
	dyn_3dim_DWORD	: ARRAY[0..ARRSIZEX, 0..ARRSIZEY, 0..ARRSIZEZ] OF DWORD;(* ~ 	(OPC : 1 : available for OPC-clients) *)
	{attribute 'OPC.UA.DA' := '1'}
	{attribute 'OPC.UA.DA.Description' := '3dim Array BOOL'}
	dyn_3dim_LWORD	: ARRAY[0..ARRSIZEX, 0..ARRSIZEY, 0..ARRSIZEZ] OF LWORD;(* ~ 	(OPC : 1 : available for OPC-clients) *)
	{attribute 'OPC.UA.DA' := '1'}
	{attribute 'OPC.UA.DA.Description' := '3dim Array BOOL'}
	dyn_3dim_R4		: ARRAY[0..ARRSIZEX, 0..ARRSIZEY, 0..ARRSIZEZ] OF REAL;(* ~ 	(OPC : 1 : available for OPC-clients) *)
	{attribute 'OPC.UA.DA' := '1'}
	{attribute 'OPC.UA.DA.Description' := '3dim Array BOOL'}
	dyn_3dim_R8		: ARRAY[0..ARRSIZEX, 0..ARRSIZEY, 0..ARRSIZEZ] OF LREAL;(* ~ 	(OPC : 1 : available for OPC-clients) *)
	{attribute 'OPC.UA.DA' := '1'}
	{attribute 'OPC.UA.DA.Description' := '3dim Array BOOL'}
	dyn_3dim_BSTR	: ARRAY[0..ARRSIZEX, 0..ARRSIZEY, 0..ARRSIZEZ] OF STRING;(* ~ 	(OPC : 1 : available for OPC-clients) *)
	{attribute 'OPC.UA.DA' := '1'}
	{attribute 'OPC.UA.DA.Description' := '3dim Array BOOL'}
	//dyn_3dim_CHAR	: ARRAY[0..ARRSIZEX, 0..ARRSIZEY, 0..ARRSIZEZ] OF CHAR;(* ~ 	(OPC : 1 : available for OPC-clients) *)
	{attribute 'OPC.UA.DA' := '1'}
	{attribute 'OPC.UA.DA.Description' := '3dim Array BOOL'}
	dyn_3dim_WSTRING : ARRAY[0..ARRSIZEX, 0..ARRSIZEY, 0..ARRSIZEZ] OF WSTRING;(* ~ 	(OPC : 1 : available for OPC-clients) *)
	{attribute 'OPC.UA.DA' := '1'}
	{attribute 'OPC.UA.DA.Description' := '3dim Array BOOL'}
	//dyn_3dim_WCHAR: ARRAY[0..ARRSIZEX, 0..ARRSIZEY, 0..ARRSIZEZ] OF WCHAR;(* ~ 	(OPC : 1 : available for OPC-clients) *)
	{attribute 'OPC.UA.DA' := '1'}
	{attribute 'OPC.UA.DA.Description' := '3dim Array BOOL'}
	dyn_3dim_DT		: ARRAY[0..ARRSIZEX, 0..ARRSIZEY, 0..ARRSIZEZ] OF DT;(* ~ 	(OPC : 1 : available for OPC-clients) *)
	{attribute 'OPC.UA.DA' := '1'}
	{attribute 'OPC.UA.DA.Description' := '3dim Array BOOL'}
	dyn_3dim_DATE 	: ARRAY[0..ARRSIZEX, 0..ARRSIZEY, 0..ARRSIZEZ] OF DATE;(* ~ 	(OPC : 1 : available for OPC-clients) *)
	{attribute 'OPC.UA.DA' := '1'}
	{attribute 'OPC.UA.DA.Description' := '3dim Array BOOL'}
	dyn_3dim_TOD	: ARRAY[0..ARRSIZEX, 0..ARRSIZEY, 0..ARRSIZEZ] OF TOD;(* ~ 	(OPC : 1 : available for OPC-clients) *)
	{attribute 'OPC.UA.DA' := '1'}
	{attribute 'OPC.UA.DA.Description' := '3dim Array BOOL'}
	dyn_3dim_TIME	: ARRAY[0..ARRSIZEX, 0..ARRSIZEY, 0..ARRSIZEZ] OF TIME;(* ~ 	(OPC : 1 : available for OPC-clients) *)
END_VAR

// ---- GVLs/GVL_nodes_static.TcGVL
VAR_GLOBAL
	//scalars
	{attribute 'OPC.UA.DA' := '1'}
	{attribute 'OPC.UA.DA.Description' := 'Scalar LINT'}
	{attribute 'OPC.UA.DA.Access' := '1'}	
	stat_scalar_BOOL	: BOOL := TRUE;
	{attribute 'OPC.UA.DA' := '1'}
	{attribute 'OPC.UA.DA.Description' := 'Scalar SINT'}
	{attribute 'OPC.UA.DA.Access' := '1'}
	stat_scalar_I1		: SINT := 1;	
	{attribute 'OPC.UA.DA' := '1'}
	{attribute 'OPC.UA.DA.Description' := 'Scalar USINT'}
	{attribute 'OPC.UA.DA.Access' := '1'}
	stat_scalar_UI1		: USINT := 1;	
	{attribute 'OPC.UA.DA' := '1'}
	{attribute 'OPC.UA.DA.Description' := 'Scalar INT'}
	{attribute 'OPC.UA.DA.Access' := '1'}
	stat_scalar_I2 		: INT := 1;		
	{attribute 'OPC.UA.DA' := '1'}
	{attribute 'OPC.UA.DA.Description' := 'Scalar UINT'}
	{attribute 'OPC.UA.DA.Access' := '1'}
	stat_scalar_UI2		: UINT := 1;	
	{attribute 'OPC.UA.DA' := '1'}
	{attribute 'OPC.UA.DA.Description' := 'Scalar DINT'}
	{attribute 'OPC.UA.DA.Access' := '1'}
	stat_scalar_I4		: DINT := 1;	
	{attribute 'OPC.UA.DA' := '1'}
	{attribute 'OPC.UA.DA.Description' := 'Scalar UDINT'}
	{attribute 'OPC.UA.DA.Access' := '1'}
	stat_scalar_UI4		: UDINT := 1;	
	{attribute 'OPC.UA.DA' := '1'}
	{attribute 'OPC.UA.DA.Description' := 'Scalar LINT'}
	{attribute 'OPC.UA.DA.Access' := '1'}
	stat_scalar_I8		: LINT := 1;	
	{attribute 'OPC.UA.DA' := '1'}
	{attribute 'OPC.UA.DA.Description' := 'Scalar ULINT'}
	{attribute 'OPC.UA.DA.Access' := '1'}
	stat_scalar_UI8		: ULINT := 1;	
	{attribute 'OPC.UA.DA' := '1'}
	{attribute 'OPC.UA.DA.Description' := 'Scalar BYTE'}
	{attribute 'OPC.UA.DA.Access' := '1'}
	stat_scalar_BYTE	: BYTE := 1;	
	{attribute 'OPC.UA.DA' := '1'}
	{attribute 'OPC.UA.DA.Description' := 'Scalar WORD'}
	{attribute 'OPC.UA.DA.Access' := '1'}
	stat_scalar_WORD	: WORD := 1;	
	{attribute 'OPC.UA.DA' := '1'}
	{attribute 'OPC.UA.DA.Description' := 'Scalar DWORD'}
	{attribute 'OPC.UA.DA.Access' := '1'}
	stat_scalar_DWORD	: DWORD := 1;	
	{attribute 'OPC.UA.DA' := '1'}
	{attribute 'OPC.UA.DA.Description' := 'Scalar LWORD'}
	{attribute 'OPC.UA.DA.Access' := '1'}
	stat_scalar_LWORD	: LWORD := 1;				
	{attribute 'OPC.UA.DA' := '1'}
	{attribute 'OPC.UA.DA.Description' := 'Scalar REAL'}
	{attribute 'OPC.UA.DA.Access' := '1'}
	stat_scalar_R4		: REAL := 1.0;				
	{attribute 'OPC.UA.DA' := '1'}
	{attribute 'OPC.UA.DA.Description' := 'Scalar LREAL'}
	{attribute 'OPC.UA.DA.Access' := '1'}
	stat_scalar_R8		: LREAL := 1.0;				
	{attribute 'OPC.UA.DA' := '1'}
	{attribute 'OPC.UA.DA.Description' := 'Scalar STRING'}
	{attribute 'OPC.UA.DA.Access' := '1'}
	stat_scalar_BSTR	: STRING := 'Hello World';
	{attribute 'OPC.UA.DA' := '1'}
	{attribute 'OPC.UA.DA.Description' := 'Scalar WSTRING'}
	{attribute 'OPC.UA.DA.Access' := '1'}
	stat_scalar_WSTRING	: WSTRING := "Hello World";
	{attribute 'OPC.UA.DA' := '1'}
	{attribute 'OPC.UA.DA.Description' := 'Scalar DT'}
	{attribute 'OPC.UA.DA.Access' := '1'}
	stat_scalar_DT		: DT;
	{attribute 'OPC.UA.DA' := '1'}
	{attribute 'OPC.UA.DA.Description' := 'Scalar DATE'}
	{attribute 'OPC.UA.DA.Access' := '1'}
	stat_scalar_DATE 	: DATE;
	{attribute 'OPC.UA.DA' := '1'}
	{attribute 'OPC.UA.DA.Description' := 'Scalar TOD'}
	{attribute 'OPC.UA.DA.Access' := '1'}
	stat_scalar_TOD		: TOD;	
	{attribute 'OPC.UA.DA' := '1'}
	{attribute 'OPC.UA.DA.Description' := 'Scalar TIME'}
	{attribute 'OPC.UA.DA.Access' := '1'}
	stat_scalar_TIME	: TIME;	

	
	//1dim
	{attribute 'OPC.UA.DA' := '1'}
	{attribute 'OPC.UA.DA.Description' := '1dim Array BOOL'}
	{attribute 'OPC.UA.DA.Access' := '1'}	
	stat_1dim_BOOL		: ARRAY[0..ARRSIZEX] OF BOOL;
	{attribute 'OPC.UA.DA' := '1'}
	{attribute 'OPC.UA.DA.Description' := '1dim Array SINT'}
	{attribute 'OPC.UA.DA.Access' := '1'}
	stat_1dim_I1		: ARRAY[0..ARRSIZEX] OF SINT;
	{attribute 'OPC.UA.DA' := '1'}
	{attribute 'OPC.UA.DA.Description' := '1dim Array USINT'}
	{attribute 'OPC.UA.DA.Access' := '1'}
	stat_1dim_UI1		: ARRAY[0..ARRSIZEX] OF USINT;
	{attribute 'OPC.UA.DA' := '1'}
	{attribute 'OPC.UA.DA.Description' := '1dim Array INT'}
	{attribute 'OPC.UA.DA.Access' := '1'}
	stat_1dim_I2 		: ARRAY[0..ARRSIZEX] OF INT;	
	{attribute 'OPC.UA.DA' := '1'}
	{attribute 'OPC.UA.DA.Description' := '1dim Array UINT'}
	{attribute 'OPC.UA.DA.Access' := '1'}
	stat_1dim_UI2		: ARRAY[0..ARRSIZEX] OF UINT;
	{attribute 'OPC.UA.DA' := '1'}
	{attribute 'OPC.UA.DA.Description' := '1dim Array DINT'}
	{attribute 'OPC.UA.DA.Access' := '1'}
	stat_1dim_I4		: ARRAY[0..ARRSIZEX] OF DINT;
	{attribute 'OPC.UA.DA' := '1'}
	{attribute 'OPC.UA.DA.Description' := '1dim Array UDINT'}
	{attribute 'OPC.UA.DA.Access' := '1'}
	stat_1dim_UI4		: ARRAY[0..ARRSIZEX] OF UDINT;
	{attribute 'OPC.UA.DA' := '1'}
	{attribute 'OPC.UA.DA.Description' := '1dim Array LINT'}
	{attribute 'OPC.UA.DA.Access' := '1'}
	stat_1dim_I8		: ARRAY[0..ARRSIZEX] OF LINT;
	{attribute 'OPC.UA.DA' := '1'}
	{attribute 'OPC.UA.DA.Description' := '1dim Array ULINT'}
	{attribute 'OPC.UA.DA.Access' := '1'}
	stat_1dim_UI8		: ARRAY[0..ARRSIZEX] OF ULINT;
	{attribute 'OPC.UA.DA' := '1'}
	{attribute 'OPC.UA.DA.Description' := '1dim Array BYTE'}
	{attribute 'OPC.UA.DA.Access' := '1'}
	stat_1dim_BYTE		: ARRAY[0..ARRSIZEX] OF BYTE;
	{attribute 'OPC.UA.DA' := '1'}
	{attribute 'OPC.UA.DA.Description' := '1dim Array WORD'}
	{attribute 'OPC.UA.DA.Access' := '1'}
	stat_1dim_WORD		: ARRAY[0..ARRSIZEX] OF WORD;
	{attribute 'OPC.UA.DA' := '1'}
	{attribute 'OPC.UA.DA.Description' := '1dim Array DWORD'}
	{attribute 'OPC.UA.DA.Access' := '1'}
	stat_1dim_DWORD		: ARRAY[0..ARRSIZEX] OF DWORD;
	{attribute 'OPC.UA.DA' := '1'}
	{attribute 'OPC.UA.DA.Description' := '1dim Array LWORD'}
	{attribute 'OPC.UA.DA.Access' := '1'}
	stat_1dim_LWORD		: ARRAY[0..ARRSIZEX] OF LWORD;
	{attribute 'OPC.UA.DA' := '1'}
	{attribute 'OPC.UA.DA.Description' := '1dim Array REAL'}
	{attribute 'OPC.UA.DA.Access' := '1'}
	stat_1dim_R4		: ARRAY[0..ARRSIZEX] OF REAL;
	{attribute 'OPC.UA.DA' := '1'}
	{attribute 'OPC.UA.DA.Description' := '1dim Array LREAL'}
	{attribute 'OPC.UA.DA.Access' := '1'}
	stat_1dim_R8		: ARRAY[0..ARRSIZEX] OF LREAL;
	{attribute 'OPC.UA.DA' := '1'}
	{attribute 'OPC.UA.DA.Description' := '1dim Array STRING'}
	{attribute 'OPC.UA.DA.Access' := '1'}
	stat_1dim_BSTR		: ARRAY[0..ARRSIZEX] OF STRING;
	{attribute 'OPC.UA.DA' := '1'}
	{attribute 'OPC.UA.DA.Description' := '1dim Array WSTRING'}
	{attribute 'OPC.UA.DA.Access' := '1'}
	stat_1dim_WSTRING	: ARRAY[0..ARRSIZEX] OF WSTRING;
	{attribute 'OPC.UA.DA' := '1'}
	{attribute 'OPC.UA.DA.Description' := '1dim Array DT'}
	{attribute 'OPC.UA.DA.Access' := '1'}
	stat_1dim_DT		: ARRAY[0..ARRSIZEX] OF DT;		
	{attribute 'OPC.UA.DA' := '1'}
	{attribute 'OPC.UA.DA.Description' := '1dim Array DATE'}
	{attribute 'OPC.UA.DA.Access' := '1'}
	stat_1dim_DATE 		: ARRAY[0..ARRSIZEX] OF DATE;	
	{attribute 'OPC.UA.DA' := '1'}
	{attribute 'OPC.UA.DA.Description' := '1dim Array TOD'}
	{attribute 'OPC.UA.DA.Access' := '1'}
	stat_1dim_TOD		: ARRAY[0..ARRSIZEX] OF TOD;	
	{attribute 'OPC.UA.DA' := '1'}
	{attribute 'OPC.UA.DA.Description' := '1dim Array TIME'}
	{attribute 'OPC.UA.DA.Access' := '1'}
	stat_1dim_TIME		: ARRAY[0..ARRSIZEX] OF TIME;	

	
	//2dim
	{attribute 'OPC.UA.DA' := '1'}
	{attribute 'OPC.UA.DA.Description' := '2dim Array BOOL'}
	stat_2dim_BOOL		: ARRAY[0..ARRSIZEX, 0..ARRSIZEY] OF BOOL;
	{attribute 'OPC.UA.DA' := '1'}
	{attribute 'OPC.UA.DA.Description' := '2dim Array SINT'}
	stat_2dim_I1		: ARRAY[0..ARRSIZEX, 0..ARRSIZEY] OF SINT;
	{attribute 'OPC.UA.DA' := '1'}
	{attribute 'OPC.UA.DA.Description' := '2dim Array USINT'}
	stat_2dim_UI1		: ARRAY[0..ARRSIZEX, 0..ARRSIZEY] OF USINT;
	{attribute 'OPC.UA.DA' := '1'}
	{attribute 'OPC.UA.DA.Description' := '2dim Array INT'}
	stat_2dim_I2 		: ARRAY[0..ARRSIZEX, 0..ARRSIZEY] OF INT;
	{attribute 'OPC.UA.DA' := '1'}
	{attribute 'OPC.UA.DA.Description' := '2dim Array UINT'}
	stat_2dim_UI2		: ARRAY[0..ARRSIZEX, 0..ARRSIZEY] OF UINT;
	{attribute 'OPC.UA.DA' := '1'}
	{attribute 'OPC.UA.DA.Description' := '2dim Array DINT'}
	stat_2dim_I4		: ARRAY[0..ARRSIZEX, 0..ARRSIZEY] OF DINT;
	{attribute 'OPC.UA.DA' := '1'}
	{attribute 'OPC.UA.DA.Description' := '2dim Array UDINT'}
	stat_2dim_UI4		: ARRAY[0..ARRSIZEX, 0..ARRSIZEY] OF UDINT;
	{attribute 'OPC.UA.DA' := '1'}
	{attribute 'OPC.UA.DA.Description' := '2dim Array LINT'}
	stat_2dim_I8		: ARRAY[0..ARRSIZEX, 0..ARRSIZEY] OF LINT;	
	{attribute 'OPC.UA.DA' := '1'}
	{attribute 'OPC.UA.DA.Description' := '2dim Array ULINT'}
	stat_2dim_UI8		: ARRAY[0..ARRSIZEX, 0..ARRSIZEY] OF ULINT;
	{attribute 'OPC.UA.DA' := '1'}
	{attribute 'OPC.UA.DA.Description' := '2dim Array BYTE'}
	stat_2dim_BYTE		: ARRAY[0..ARRSIZEX, 0..ARRSIZEY] OF BYTE;	
	{attribute 'OPC.UA.DA' := '1'}
	{attribute 'OPC.UA.DA.Description' := '2dim Array WORD'}
	stat_2dim_WORD		: ARRAY[0..ARRSIZEX, 0..ARRSIZEY] OF WORD;	
	{attribute 'OPC.UA.DA' := '1'}
	{attribute 'OPC.UA.DA.Description' := '2dim Array DWORD'}
	stat_2dim_DWORD		: ARRAY[0..ARRSIZEX, 0..ARRSIZEY] OF DWORD;	
	{attribute 'OPC.UA.DA' := '1'}
	{attribute 'OPC.UA.DA.Description' := '2dim Array LWORD'}
	stat_2dim_LWORD		: ARRAY[0..ARRSIZEX, 0..ARRSIZEY] OF LWORD;
	{attribute 'OPC.UA.DA' := '1'}
	{attribute 'OPC.UA.DA.Description' := '2dim Array REAL'}
	stat_2dim_R4		: ARRAY[0..ARRSIZEX, 0..ARRSIZEY] OF REAL;
	{attribute 'OPC.UA.DA' := '1'}
	{attribute 'OPC.UA.DA.Description' := '2dim Array LREAL'}
	stat_2dim_R8		: ARRAY[0..ARRSIZEX, 0..ARRSIZEY] OF LREAL;
	{attribute 'OPC.UA.DA' := '1'}
	{attribute 'OPC.UA.DA.Description' := '2dim Array STRING'}
	stat_2dim_BSTR		: ARRAY[0..ARRSIZEX, 0..ARRSIZEY] OF STRING;
	{attribute 'OPC.UA.DA' := '1'}
	{attribute 'OPC.UA.DA.Description' := '2dim Array WSTRING'}
	stat_2dim_WSTRING	: ARRAY[0..ARRSIZEX, 0..ARRSIZEY] OF WSTRING;
	{attribute 'OPC.UA.DA' := '1'}
	{attribute 'OPC.UA.DA.Description' := '2dim Array DT'}
	stat_2dim_DT		: ARRAY[0..ARRSIZEX, 0..ARRSIZEY] OF DT;
	{attribute 'OPC.UA.DA' := '1'}
	{attribute 'OPC.UA.DA.Description' := '2dim Array DATE'}
	stat_2dim_DATE	 	: ARRAY[0..ARRSIZEX, 0..ARRSIZEY] OF DATE;
	{attribute 'OPC.UA.DA' := '1'}
	{attribute 'OPC.UA.DA.Description' := '2dim Array TOD'}
	stat_2dim_TOD		: ARRAY[0..ARRSIZEX, 0..ARRSIZEY] OF TOD;
	{attribute 'OPC.UA.DA' := '1'}
	{attribute 'OPC.UA.DA.Description' := '2dim Array TIME'}
	stat_2dim_TIME		: ARRAY[0..ARRSIZEX, 0..ARRSIZEY] OF TIME;

	//3dim
	{attribute 'OPC.UA.DA' := '1'}
	{attribute 'OPC.UA.DA.Description' := '3dim Array BOOL'}
	stat_3dim_BOOL		: ARRAY[0..ARRSIZEX, 0..ARRSIZEY, 0..ARRSIZEZ] OF BOOL;
	{attribute 'OPC.UA.DA' := '1'}
	{attribute 'OPC.UA.DA.Description' := '2dim Array SINT'}
	stat_3dim_I1		: ARRAY[0..ARRSIZEX, 0..ARRSIZEY, 0..ARRSIZEZ] OF SINT;
	{attribute 'OPC.UA.DA' := '1'}
	{attribute 'OPC.UA.DA.Description' := '2dim Array USINT'}
	stat_3dim_UI1		: ARRAY[0..ARRSIZEX, 0..ARRSIZEY, 0..ARRSIZEZ] OF USINT;
	{attribute 'OPC.UA.DA' := '1'}
	{attribute 'OPC.UA.DA.Description' := '2dim Array INT'}
	stat_3dim_I2 		: ARRAY[0..ARRSIZEX, 0..ARRSIZEY, 0..ARRSIZEZ] OF INT;
	{attribute 'OPC.UA.DA' := '1'}
	{attribute 'OPC.UA.DA.Description' := '2dim Array UINT'}
	stat_3dim_UI2		: ARRAY[0..ARRSIZEX, 0..ARRSIZEY, 0..ARRSIZEZ] OF UINT;
	{attribute 'OPC.UA.DA' := '1'}
	{attribute 'OPC.UA.DA.Description' := '2dim Array DINT'}
	stat_3dim_I4		: ARRAY[0..ARRSIZEX, 0..ARRSIZEY, 0..ARRSIZEZ] OF DINT;
	{attribute 'OPC.UA.DA' := '1'}
	{attribute 'OPC.UA.DA.Description' := '2dim Array UDINT'}
	stat_3dim_UI4		: ARRAY[0..ARRSIZEX, 0..ARRSIZEY, 0..ARRSIZEZ] OF UDINT;
	{attribute 'OPC.UA.DA' := '1'}
	{attribute 'OPC.UA.DA.Description' := '2dim Array LINT'}
	stat_3dim_I8		: ARRAY[0..ARRSIZEX, 0..ARRSIZEY, 0..ARRSIZEZ] OF LINT;
	{attribute 'OPC.UA.DA' := '1'}
	{attribute 'OPC.UA.DA.Description' := '2dim Array ULINT'}
	stat_3dim_UI8		: ARRAY[0..ARRSIZEX, 0..ARRSIZEY, 0..ARRSIZEZ] OF ULINT;
	{attribute 'OPC.UA.DA' := '1'}
	{attribute 'OPC.UA.DA.Description' := '2dim Array BYTE'}
	stat_3dim_BYTE		: ARRAY[0..ARRSIZEX, 0..ARRSIZEY, 0..ARRSIZEZ] OF BYTE;
	{attribute 'OPC.UA.DA' := '1'}
	{attribute 'OPC.UA.DA.Description' := '2dim Array WORD'}
	stat_3dim_WORD		: ARRAY[0..ARRSIZEX, 0..ARRSIZEY, 0..ARRSIZEZ] OF WORD;
	{attribute 'OPC.UA.DA' := '1'}
	{attribute 'OPC.UA.DA.Description' := '2dim Array DWORD'}
	stat_3dim_DWORD		: ARRAY[0..ARRSIZEX, 0..ARRSIZEY, 0..ARRSIZEZ] OF DWORD;
	{attribute 'OPC.UA.DA' := '1'}
	{attribute 'OPC.UA.DA.Description' := '2dim Array LWORD'}
	stat_3dim_LWORD		: ARRAY[0..ARRSIZEX, 0..ARRSIZEY, 0..ARRSIZEZ] OF LWORD;
	{attribute 'OPC.UA.DA' := '1'}
	{attribute 'OPC.UA.DA.Description' := '2dim Array REAL'}
	stat_3dim_R4		: ARRAY[0..ARRSIZEX, 0..ARRSIZEY, 0..ARRSIZEZ] OF REAL;	
	{attribute 'OPC.UA.DA' := '1'}
	{attribute 'OPC.UA.DA.Description' := '2dim Array LREAL'}
	stat_3dim_R8		: ARRAY[0..ARRSIZEX, 0..ARRSIZEY, 0..ARRSIZEZ] OF LREAL;
	{attribute 'OPC.UA.DA' := '1'}
	{attribute 'OPC.UA.DA.Description' := '2dim Array STRING'}
	stat_3dim_BSTR		: ARRAY[0..ARRSIZEX, 0..ARRSIZEY, 0..ARRSIZEZ] OF STRING;
	{attribute 'OPC.UA.DA' := '1'}
	{attribute 'OPC.UA.DA.Description' := '2dim Array WSTRING'}
	stat_3dim_WSTRING 	: ARRAY[0..ARRSIZEX, 0..ARRSIZEY, 0..ARRSIZEZ] OF WSTRING;
	{attribute 'OPC.UA.DA' := '1'}
	{attribute 'OPC.UA.DA.Description' := '2dim Array DT'}
	stat_3dim_DT		: ARRAY[0..ARRSIZEX, 0..ARRSIZEY, 0..ARRSIZEZ] OF DT;
	{attribute 'OPC.UA.DA' := '1'}
	{attribute 'OPC.UA.DA.Description' := '2dim Array DATE'}
	stat_3dim_DATE 		: ARRAY[0..ARRSIZEX, 0..ARRSIZEY, 0..ARRSIZEZ] OF DATE;
	{attribute 'OPC.UA.DA' := '1'}
	{attribute 'OPC.UA.DA.Description' := '2dim Array TOD'}
	stat_3dim_TOD		: ARRAY[0..ARRSIZEX, 0..ARRSIZEY, 0..ARRSIZEZ] OF TOD;	
	{attribute 'OPC.UA.DA' := '1'}
	{attribute 'OPC.UA.DA.Description' := '2dim Array TIME'}
	stat_3dim_TIME		: ARRAY[0..ARRSIZEX, 0..ARRSIZEY, 0..ARRSIZEZ] OF TIME;

	
	// Scalars writeable
	{attribute 'OPC.UA.DA' := '1'}
	{attribute 'OPC.UA.DA.Description' := 'Scalar LINT'}	
	stat_scalar_BOOL_writeable	: BOOL := TRUE;
	{attribute 'OPC.UA.DA' := '1'}
	{attribute 'OPC.UA.DA.Description' := 'Scalar SINT'}
	stat_scalar_I1_writeable		: SINT := 1;	
	{attribute 'OPC.UA.DA' := '1'}
	{attribute 'OPC.UA.DA.Description' := 'Scalar USINT'}
	stat_scalar_UI1_writeable		: USINT := 1;	
	{attribute 'OPC.UA.DA' := '1'}
	{attribute 'OPC.UA.DA.Description' := 'Scalar INT'}
	stat_scalar_I2_writeable 		: INT := 1;		
	{attribute 'OPC.UA.DA' := '1'}
	{attribute 'OPC.UA.DA.Description' := 'Scalar UINT'}
	stat_scalar_UI2_writeable		: UINT := 1;	
	{attribute 'OPC.UA.DA' := '1'}
	{attribute 'OPC.UA.DA.Description' := 'Scalar DINT'}
	stat_scalar_I4_writeable		: DINT := 1;	
	{attribute 'OPC.UA.DA' := '1'}
	{attribute 'OPC.UA.DA.Description' := 'Scalar UDINT'}
	stat_scalar_UI4_writeable		: UDINT := 1;	
	{attribute 'OPC.UA.DA' := '1'}
	{attribute 'OPC.UA.DA.Description' := 'Scalar LINT'}
	stat_scalar_I8_writeable		: LINT := 1;	
	{attribute 'OPC.UA.DA' := '1'}
	{attribute 'OPC.UA.DA.Description' := 'Scalar ULINT'}
	stat_scalar_UI8_writeable		: ULINT := 1;	
	{attribute 'OPC.UA.DA' := '1'}
	{attribute 'OPC.UA.DA.Description' := 'Scalar BYTE'}
	stat_scalar_BYTE_writeable	: BYTE := 1;	
	{attribute 'OPC.UA.DA' := '1'}
	{attribute 'OPC.UA.DA.Description' := 'Scalar WORD'}
	stat_scalar_WORD_writeable	: WORD := 1;	
	{attribute 'OPC.UA.DA' := '1'}
	{attribute 'OPC.UA.DA.Description' := 'Scalar DWORD'}
	stat_scalar_DWORD_writeable	: DWORD := 1;	
	{attribute 'OPC.UA.DA' := '1'}
	{attribute 'OPC.UA.DA.Description' := 'Scalar LWORD'}
	stat_scalar_LWORD_writeable	: LWORD := 1;				
	{attribute 'OPC.UA.DA' := '1'}
	{attribute 'OPC.UA.DA.Description' := 'Scalar REAL'}
	stat_scalar_R4_writeable		: REAL := 1.0;				
	{attribute 'OPC.UA.DA' := '1'}
	{attribute 'OPC.UA.DA.Description' := 'Scalar LREAL'}
	stat_scalar_R8_writeable		: LREAL := 1.0;				
	{attribute 'OPC.UA.DA' := '1'}
	{attribute 'OPC.UA.DA.Description' := 'Scalar STRING'}
	stat_scalar_BSTR_writeable	: STRING := 'Hello World';
	{attribute 'OPC.UA.DA' := '1'}
	{attribute 'OPC.UA.DA.Description' := 'Scalar WSTRING'}
	stat_scalar_WSTRING_writeable	: WSTRING := "Hello World";
	{attribute 'OPC.UA.DA' := '1'}
	{attribute 'OPC.UA.DA.Description' := 'Scalar DT'}
	stat_scalar_DT_writeable		: DT;
	{attribute 'OPC.UA.DA' := '1'}
	{attribute 'OPC.UA.DA.Description' := 'Scalar DATE'}
	stat_scalar_DATE_writeable 	: DATE;
	{attribute 'OPC.UA.DA' := '1'}
	{attribute 'OPC.UA.DA.Description' := 'Scalar TOD'}
	stat_scalar_TOD_writeable		: TOD;	
	{attribute 'OPC.UA.DA' := '1'}
	{attribute 'OPC.UA.DA.Description' := 'Scalar TIME'}
	stat_scalar_TIME_writeable	: TIME;	

	
	//1dim
	{attribute 'OPC.UA.DA' := '1'}
	{attribute 'OPC.UA.DA.Description' := '1dim Array BOOL'}	
	stat_1dim_BOOL_writeable		: ARRAY[0..ARRSIZEX] OF BOOL;
	{attribute 'OPC.UA.DA' := '1'}
	{attribute 'OPC.UA.DA.Description' := '1dim Array SINT'}
	stat_1dim_I1_writeable		: ARRAY[0..ARRSIZEX] OF SINT;
	{attribute 'OPC.UA.DA' := '1'}
	{attribute 'OPC.UA.DA.Description' := '1dim Array USINT'}
	stat_1dim_UI1_writeable		: ARRAY[0..ARRSIZEX] OF USINT;
	{attribute 'OPC.UA.DA' := '1'}
	{attribute 'OPC.UA.DA.Description' := '1dim Array INT'}
	stat_1dim_I2_writeable 		: ARRAY[0..ARRSIZEX] OF INT;	
	{attribute 'OPC.UA.DA' := '1'}
	{attribute 'OPC.UA.DA.Description' := '1dim Array UINT'}
	stat_1dim_UI2_writeable		: ARRAY[0..ARRSIZEX] OF UINT;
	{attribute 'OPC.UA.DA' := '1'}
	{attribute 'OPC.UA.DA.Description' := '1dim Array DINT'}
	stat_1dim_I4_writeable		: ARRAY[0..ARRSIZEX] OF DINT;
	{attribute 'OPC.UA.DA' := '1'}
	{attribute 'OPC.UA.DA.Description' := '1dim Array UDINT'}
	stat_1dim_UI4_writeable		: ARRAY[0..ARRSIZEX] OF UDINT;
	{attribute 'OPC.UA.DA' := '1'}
	{attribute 'OPC.UA.DA.Description' := '1dim Array LINT'}
	stat_1dim_I8_writeable		: ARRAY[0..ARRSIZEX] OF LINT;
	{attribute 'OPC.UA.DA' := '1'}
	{attribute 'OPC.UA.DA.Description' := '1dim Array ULINT'}
	stat_1dim_UI8_writeable		: ARRAY[0..ARRSIZEX] OF ULINT;
	{attribute 'OPC.UA.DA' := '1'}
	{attribute 'OPC.UA.DA.Description' := '1dim Array BYTE'}
	stat_1dim_BYTE_writeable		: ARRAY[0..ARRSIZEX] OF BYTE;
	{attribute 'OPC.UA.DA' := '1'}
	{attribute 'OPC.UA.DA.Description' := '1dim Array WORD'}
	stat_1dim_WORD_writeable		: ARRAY[0..ARRSIZEX] OF WORD;
	{attribute 'OPC.UA.DA' := '1'}
	{attribute 'OPC.UA.DA.Description' := '1dim Array DWORD'}
	stat_1dim_DWORD_writeable		: ARRAY[0..ARRSIZEX] OF DWORD;
	{attribute 'OPC.UA.DA' := '1'}
	{attribute 'OPC.UA.DA.Description' := '1dim Array LWORD'}
	stat_1dim_LWORD_writeable		: ARRAY[0..ARRSIZEX] OF LWORD;
	{attribute 'OPC.UA.DA' := '1'}
	{attribute 'OPC.UA.DA.Description' := '1dim Array REAL'}
	stat_1dim_R4_writeable		: ARRAY[0..ARRSIZEX] OF REAL;
	{attribute 'OPC.UA.DA' := '1'}
	{attribute 'OPC.UA.DA.Description' := '1dim Array LREAL'}
	stat_1dim_R8_writeable		: ARRAY[0..ARRSIZEX] OF LREAL;
	{attribute 'OPC.UA.DA' := '1'}
	{attribute 'OPC.UA.DA.Description' := '1dim Array STRING'}
	stat_1dim_BSTR_writeable		: ARRAY[0..ARRSIZEX] OF STRING;
	{attribute 'OPC.UA.DA' := '1'}
	{attribute 'OPC.UA.DA.Description' := '1dim Array WSTRING'}
	stat_1dim_WSTRING_writeable	: ARRAY[0..ARRSIZEX] OF WSTRING;
	{attribute 'OPC.UA.DA' := '1'}
	{attribute 'OPC.UA.DA.Description' := '1dim Array DT'}
	stat_1dim_DT_writeable		: ARRAY[0..ARRSIZEX] OF DT;		
	{attribute 'OPC.UA.DA' := '1'}
	{attribute 'OPC.UA.DA.Description' := '1dim Array DATE'}
	stat_1dim_DATE_writeable 		: ARRAY[0..ARRSIZEX] OF DATE;	
	{attribute 'OPC.UA.DA' := '1'}
	{attribute 'OPC.UA.DA.Description' := '1dim Array TOD'}
	stat_1dim_TOD_writeable		: ARRAY[0..ARRSIZEX] OF TOD;	
	{attribute 'OPC.UA.DA' := '1'}
	{attribute 'OPC.UA.DA.Description' := '1dim Array TIME'}
	stat_1dim_TIME_writeable		: ARRAY[0..ARRSIZEX] OF TIME;		
END_VAR

// ---- POUs/Methods/FB_Methods.TcPOU
FUNCTION_BLOCK FB_Methods
VAR
	count : LREAL;
END_VAR

{attribute 'TcRpcEnable'}
{attribute 'OPC.UA.DA.Description' := 'Returns array of INT'}
METHOD M_Array_1 : ARRAY[0..2] OF INT
VAR_INPUT
END_VAR
VAR
	aTest : ARRAY[0..2] OF INT;
END_VAR
aTest[0] := 1;
aTest[1] := 2;
aTest[2] := 3;
M_Array_1 := aTest;
END_METHOD

{attribute 'TcRpcEnable'}
{attribute 'OPC.UA.DA.Description' := 'Returns simple complex type'}
METHOD M_Complex_1 : ST_Complex_1
count :=count+1;
M_Complex_1.a := 1;
M_Complex_1.b := 2;
END_METHOD

{attribute 'TcRpcEnable'}
{attribute 'OPC.UA.DA.Description' := 'InOut argument is a simple complex type'}
METHOD M_Complex_2 : ST_Complex_1
VAR_INPUT
	in : ST_Complex_1;
END_VAR
count :=count+1;
M_Complex_2.a := in.a + 1;
M_Complex_2.b := in.b + 1;
END_METHOD

END_FUNCTION_BLOCK

// ---- POUs/Programs/PRG_Dynamic.TcPOU
PROGRAM PRG_Dynamic
VAR
	k: INT;
	l: INT;
	m: INT;
	t: INT;
	
	timer_1s : TON := (PT:=T#1S);
	timer_30s : TON := (PT:=T#30S);
	timer_100ms : TON := (PT:=T#100MS);
	
	idxEndChar :INT := 0;
	idxStartChar :INT := 1;
	
	nTextMode :INT := 0;	
	
	sWordsU : WSTRING :=  "Hello OpcUA. Greetings from BECKHOFF AUTOMATION GmbH";
	sWordsA : STRING :=  'Hello OpcUA. Greetings from BECKHOFF AUTOMATION GmbH';	
END_VAR

Settings.UpdateTimer(IN:=TRUE);
timer_100ms(IN:=TRUE);
timer_1s(IN:=TRUE);
timer_30s(IN:=TRUE);

IF( timer_100ms.Q ) THEN 
	CASE nTextMode OF
		0:		
			idxStartChar := 1;
			idxEndChar :=idxEndChar+1;
			IF( idxEndChar > LEN( sWordsA ))THEN
				idxEndChar := LEN( sWordsA );
				idxStartChar :=1;	
				nTextMode := 1;
			END_IF
		1:
			idxEndChar := LEN( sWordsA );
			idxStartChar := idxStartChar+1;
			IF( idxStartChar >= LEN( sWordsA ))THEN
				idxStartChar := 1;	
				idxEndChar := 0	;		
				nTextMode := 0;
			END_IF
	END_CASE	 
END_IF

IF Settings.UpdateTimer.Q THEN
	Settings.UpdateTimer(IN:=FALSE);
	
	(* Update variables with new values *)
	GVL_nodes_dynamic.dyn_scalar_BOOL 	:= NOT GVL_nodes_dynamic.dyn_scalar_BOOL;
	GVL_nodes_dynamic.dyn_scalar_I1 		:= GVL_nodes_dynamic.dyn_scalar_I1  +1;
	GVL_nodes_dynamic.dyn_scalar_UI1 		:= GVL_nodes_dynamic.dyn_scalar_UI1 +1;
	GVL_nodes_dynamic.dyn_scalar_I2		:= GVL_nodes_dynamic.dyn_scalar_I2  +1;
	GVL_nodes_dynamic.dyn_scalar_UI2		:= GVL_nodes_dynamic.dyn_scalar_UI2 +1;
	GVL_nodes_dynamic.dyn_scalar_I4		:= GVL_nodes_dynamic.dyn_scalar_I4  +1;
	GVL_nodes_dynamic.dyn_scalar_UI4		:= GVL_nodes_dynamic.dyn_scalar_UI4 +1;
	GVL_nodes_dynamic.dyn_scalar_I8		:= GVL_nodes_dynamic.dyn_scalar_I8  +1;
	GVL_nodes_dynamic.dyn_scalar_UI8		:= GVL_nodes_dynamic.dyn_scalar_UI8 +1;
	GVL_nodes_dynamic.dyn_scalar_BYTE 	:= GVL_nodes_dynamic.dyn_scalar_BYTE +1;
	GVL_nodes_dynamic.dyn_scalar_WORD		:= GVL_nodes_dynamic.dyn_scalar_WORD +1;
	GVL_nodes_dynamic.dyn_scalar_DWORD	:= GVL_nodes_dynamic.dyn_scalar_DWORD+1;
	GVL_nodes_dynamic.dyn_scalar_LWORD    := GVL_nodes_dynamic.dyn_scalar_LWORD+1;
	GVL_nodes_dynamic.dyn_scalar_R4       := GVL_nodes_dynamic.dyn_scalar_R4+0.1;
	GVL_nodes_dynamic.dyn_scalar_R8		:= GVL_nodes_dynamic.dyn_scalar_R8+0.1;
	IF( timer_100ms.Q ) THEN 	
		GVL_nodes_dynamic.dyn_scalar_BSTR	:=  MID(STR:=sWordsA, POS:=idxStartChar, LEN:=idxEndChar); //CONCAT(GVL_dynamic_.dyn_scalar_BSTR, MID(sWordsA, 1,idxWords) );
		GVL_nodes_dynamic.dyn_scalar_WSTRING  :=  WMID(STR:=sWordsU, POS:=idxStartChar, LEN:=idxEndChar);// WCONCAT(GVL_dynamic_.dyn_scalar_WSTRING,WMID(sWordsU,1,idxWords));
	END_IF
	GVL_nodes_dynamic.dyn_scalar_DT		:= GVL_nodes_dynamic.dyn_scalar_DT 	+ T#1S;
	GVL_nodes_dynamic.dyn_scalar_DATE 	:= GVL_nodes_dynamic.dyn_scalar_DATE  + T#1S;
	GVL_nodes_dynamic.dyn_scalar_TOD		:= GVL_nodes_dynamic.dyn_scalar_TOD   + T#1S;
	GVL_nodes_dynamic.dyn_scalar_TIME		:= GVL_nodes_dynamic.dyn_scalar_TIME  + T#1S;
	
	FOR k:= 0 TO ARRSIZEHUGE DO
		GVL_nodes_dynamic.dyn_1dim_I1_Huge[k] 	:= GVL_nodes_dynamic.dyn_1dim_I1_Huge[k]  +1;
		GVL_nodes_dynamic.dyn_1dim_I4_Huge[k] 	:= GVL_nodes_dynamic.dyn_1dim_I4_Huge[k]  +1;
	END_FOR
	
	FOR k:= 0 TO ARRSIZEX DO
		GVL_nodes_dynamic.dyn_1dim_BOOL[k] 	:= NOT GVL_nodes_dynamic.dyn_1dim_BOOL[k];
		GVL_nodes_dynamic.dyn_1dim_I1[k] 		:= GVL_nodes_dynamic.dyn_1dim_I1[k]  +1;
		GVL_nodes_dynamic.dyn_1dim_UI1[k]		:= GVL_nodes_dynamic.dyn_1dim_UI1[k] +1;
		GVL_nodes_dynamic.dyn_1dim_I2[k]		:= GVL_nodes_dynamic.dyn_1dim_I2[k]  +1;
		GVL_nodes_dynamic.dyn_1dim_UI2[k]		:= GVL_nodes_dynamic.dyn_1dim_UI2[k] +1;
		GVL_nodes_dynamic.dyn_1dim_I4[k]		:= GVL_nodes_dynamic.dyn_1dim_I4[k]  +1;
		GVL_nodes_dynamic.dyn_1dim_UI4[k]		:= GVL_nodes_dynamic.dyn_1dim_UI4[k] +1;
		GVL_nodes_dynamic.dyn_1dim_I8[k]		:= GVL_nodes_dynamic.dyn_1dim_I8[k]  +1;
		GVL_nodes_dynamic.dyn_1dim_UI8[k]		:= GVL_nodes_dynamic.dyn_1dim_UI8[k] +1;
		GVL_nodes_dynamic.dyn_1dim_BYTE[k] 	:= GVL_nodes_dynamic.dyn_1dim_BYTE[k] +1;
		GVL_nodes_dynamic.dyn_1dim_WORD[k]	:= GVL_nodes_dynamic.dyn_1dim_WORD[k] +1;
		GVL_nodes_dynamic.dyn_1dim_DWORD[k]	:= GVL_nodes_dynamic.dyn_1dim_DWORD[k]+1;
		GVL_nodes_dynamic.dyn_1dim_LWORD[k]   := GVL_nodes_dynamic.dyn_1dim_LWORD[k]+1;
		GVL_nodes_dynamic.dyn_1dim_R4[k]      := GVL_nodes_dynamic.dyn_1dim_R4[k]+0.1;
		GVL_nodes_dynamic.dyn_1dim_R8[k]		:= GVL_nodes_dynamic.dyn_1dim_R8[k]+0.1;
		IF( timer_100ms.Q ) THEN 	
			GVL_nodes_dynamic.dyn_1dim_BSTR[k]	:=  MID(STR:=sWordsA, POS:=idxStartChar, LEN:=idxEndChar); //CONCAT(GVL_dynamic_.dyn_scalar_BSTR, MID(sWordsA, 1,idxWords) );
			GVL_nodes_dynamic.dyn_1dim_WSTRING[k]  :=  WMID(STR:=sWordsU, POS:=idxStartChar, LEN:=idxEndChar);// WCONCAT(GVL_dynamic_.dyn_scalar_WSTRING,WMID(sWordsU,1,idxWords));
		END_IF
		GVL_nodes_dynamic.dyn_1dim_DT[k]		:= GVL_nodes_dynamic.dyn_1dim_DT[k] 	+ T#1S;
		GVL_nodes_dynamic.dyn_1dim_DATE[k] 	:= GVL_nodes_dynamic.dyn_1dim_DATE[k]  + T#1S;
		GVL_nodes_dynamic.dyn_1dim_TOD[k]		:= GVL_nodes_dynamic.dyn_1dim_TOD[k]   + T#1S;
		GVL_nodes_dynamic.dyn_1dim_TIME[k]	:= GVL_nodes_dynamic.dyn_1dim_TIME[k]  + T#1S;
	END_FOR;
	
	FOR l:= 0 TO ARRSIZEY DO
		FOR k:= 0 TO ARRSIZEX DO
			GVL_nodes_dynamic.dyn_2dim_BOOL[k,l] 		:= NOT GVL_nodes_dynamic.dyn_2dim_BOOL[k,l];
			GVL_nodes_dynamic.dyn_2dim_I1[k,l] 		:= GVL_nodes_dynamic.dyn_2dim_I1[k,l]  +1;
			GVL_nodes_dynamic.dyn_2dim_UI1[k,l]		:= GVL_nodes_dynamic.dyn_2dim_UI1[k,l] +1;
			GVL_nodes_dynamic.dyn_2dim_I2[k,l]		:= GVL_nodes_dynamic.dyn_2dim_I2[k,l]  +1;
			GVL_nodes_dynamic.dyn_2dim_UI2[k,l]		:= GVL_nodes_dynamic.dyn_2dim_UI2[k,l] +1;
			GVL_nodes_dynamic.dyn_2dim_I4[k,l]		:= GVL_nodes_dynamic.dyn_2dim_I4[k,l]  +1;
			GVL_nodes_dynamic.dyn_2dim_UI4[k,l]		:= GVL_nodes_dynamic.dyn_2dim_UI4[k,l] +1;
			GVL_nodes_dynamic.dyn_2dim_I8[k,l]		:= GVL_nodes_dynamic.dyn_2dim_I8[k,l]  +1;
			GVL_nodes_dynamic.dyn_2dim_UI8[k,l]		:= GVL_nodes_dynamic.dyn_2dim_UI8[k,l] +1;
			GVL_nodes_dynamic.dyn_2dim_BYTE[k,l] 		:= GVL_nodes_dynamic.dyn_2dim_BYTE[k,l] +1;
			GVL_nodes_dynamic.dyn_2dim_WORD[k,l]		:= GVL_nodes_dynamic.dyn_2dim_WORD[k,l] +1;
			GVL_nodes_dynamic.dyn_2dim_DWORD[k,l]		:= GVL_nodes_dynamic.dyn_2dim_DWORD[k,l]+1;
			GVL_nodes_dynamic.dyn_2dim_LWORD[k,l]    	:= GVL_nodes_dynamic.dyn_2dim_LWORD[k,l]+1;
			GVL_nodes_dynamic.dyn_2dim_R4[k,l]       	:= GVL_nodes_dynamic.dyn_2dim_R4[k,l]+0.1;
			GVL_nodes_dynamic.dyn_2dim_R8[k,l]		:= GVL_nodes_dynamic.dyn_2dim_R8[k,l]+0.1;
			IF( timer_100ms.Q ) THEN 	
				GVL_nodes_dynamic.dyn_2dim_BSTR[k,l]	:=  MID(STR:=sWordsA, POS:=idxStartChar, LEN:=idxEndChar); //CONCAT(GVL_dynamic_.dyn_scalar_BSTR, MID(sWordsA, 1,idxWords) );
				GVL_nodes_dynamic.dyn_2dim_WSTRING[k,l]  :=  WMID(STR:=sWordsU, POS:=idxStartChar, LEN:=idxEndChar);// WCONCAT(GVL_dynamic_.dyn_scalar_WSTRING,WMID(sWordsU,1,idxWords));
			END_IF
			GVL_nodes_dynamic.dyn_2dim_DT[k,l]		:= GVL_nodes_dynamic.dyn_2dim_DT[k,l] 	+ T#1S;
			GVL_nodes_dynamic.dyn_2dim_DATE[k,l] 	:= GVL_nodes_dynamic.dyn_2dim_DATE[k,l]  + T#1S;
			GVL_nodes_dynamic.dyn_2dim_TOD[k,l]	:= GVL_nodes_dynamic.dyn_2dim_TOD[k,l]   + T#1S;
			GVL_nodes_dynamic.dyn_2dim_TIME[k,l]		:= GVL_nodes_dynamic.dyn_2dim_TIME[k,l] + T#1S;
		END_FOR;
	END_FOR;
	
	FOR m:= 0 TO ARRSIZEY DO
		FOR l:= 0 TO ARRSIZEY DO
			FOR k:= 0 TO ARRSIZEX DO
				GVL_nodes_dynamic.dyn_3dim_BOOL[k,l,m] 		:= NOT GVL_nodes_dynamic.dyn_3dim_BOOL[k,l,m];
				GVL_nodes_dynamic.dyn_3dim_I1[k,l,m] 		:= GVL_nodes_dynamic.dyn_3dim_I1[k,l,m]  +1;
				GVL_nodes_dynamic.dyn_3dim_UI1[k,l,m]		:= GVL_nodes_dynamic.dyn_3dim_UI1[k,l,m] +1;
				GVL_nodes_dynamic.dyn_3dim_I2[k,l,m]		:= GVL_nodes_dynamic.dyn_3dim_I2[k,l,m]  +1;
				GVL_nodes_dynamic.dyn_3dim_UI2[k,l,m]		:= GVL_nodes_dynamic.dyn_3dim_UI2[k,l,m] +1;
				GVL_nodes_dynamic.dyn_3dim_I4[k,l,m]		:= GVL_nodes_dynamic.dyn_3dim_I4[k,l,m]  +1;
				GVL_nodes_dynamic.dyn_3dim_UI4[k,l,m]		:= GVL_nodes_dynamic.dyn_3dim_UI4[k,l,m] +1;
				GVL_nodes_dynamic.dyn_3dim_I8[k,l,m]		:= GVL_nodes_dynamic.dyn_3dim_I8[k,l,m]  +1;
				GVL_nodes_dynamic.dyn_3dim_UI8[k,l,m]		:= GVL_nodes_dynamic.dyn_3dim_UI8[k,l,m] +1;
				GVL_nodes_dynamic.dyn_3dim_BYTE[k,l,m] 		:= GVL_nodes_dynamic.dyn_3dim_BYTE[k,l,m] +1;
				GVL_nodes_dynamic.dyn_3dim_WORD[k,l,m]		:= GVL_nodes_dynamic.dyn_3dim_WORD[k,l,m] +1;
				GVL_nodes_dynamic.dyn_3dim_DWORD[k,l,m]		:= GVL_nodes_dynamic.dyn_3dim_DWORD[k,l,m]+1;
				GVL_nodes_dynamic.dyn_3dim_LWORD[k,l,m]    	:= GVL_nodes_dynamic.dyn_3dim_LWORD[k,l,m]+1;
				GVL_nodes_dynamic.dyn_3dim_R4[k,l,m]       	:= GVL_nodes_dynamic.dyn_3dim_R4[k,l,m]+0.1;
				GVL_nodes_dynamic.dyn_3dim_R8[k,l,m]		:= GVL_nodes_dynamic.dyn_3dim_R8[k,l,m]+0.1;
				IF( timer_100ms.Q ) THEN 	
					GVL_nodes_dynamic.dyn_3dim_BSTR[k,l,m]	:=  MID(STR:=sWordsA, POS:=idxStartChar, LEN:=idxEndChar); //CONCAT(GVL_dynamic_.dyn_scalar_BSTR, MID(sWordsA, 1,idxWords) );
					GVL_nodes_dynamic.dyn_3dim_WSTRING[k,l,m]  :=  WMID(STR:=sWordsU, POS:=idxStartChar, LEN:=idxEndChar);// WCONCAT(GVL_dynamic_.dyn_scalar_WSTRING,WMID(sWordsU,1,idxWords));
				END_IF	
				GVL_nodes_dynamic.dyn_3dim_DT[k,l,m]		:= GVL_nodes_dynamic.dyn_3dim_DT[k,l,m] 	+ T#1S;
				GVL_nodes_dynamic.dyn_3dim_DATE[k,l,m] 	:= GVL_nodes_dynamic.dyn_3dim_DATE[k,l,m]  + T#1S;
				GVL_nodes_dynamic.dyn_3dim_TOD[k,l,m]	:= GVL_nodes_dynamic.dyn_3dim_TOD[k,l,m]   + T#1S;
				GVL_nodes_dynamic.dyn_3dim_TIME[k,l,m]		:= GVL_nodes_dynamic.dyn_3dim_TIME[k,l,m] + T#1S;
			END_FOR;
		END_FOR;
	END_FOR;
END_IF

(*
-----------------------------------------------------------------------------------------------------
Historical Access
-----------------------------------------------------------------------------------------------------					
*)
t := t + 1;
o := o + 0.001;

sinu := SIN(o);
cosinu := COS(o);

i:=i+1;
Ts:=128*10;

phi:=t/Ts;
Cosinus_Half:=COS(PI*t/(2*Ts));

Sinus_VerySlow:=COS(1*PI*(t)/Ts);
Sinus_Slow1:=COS(4*PI* (t+Ts/4+phi)/Ts);
Sinus_Slow2:= 0.000001*COS(4*PI* (t+Ts/3+phi)/Ts);
Sinus_Fast:=COS(12*PI*t/Ts);
Sinus_SqFast:=Sinus_Fast* Sinus_Slow1;
Sinus_SqSlow:=Sinus_VerySlow*Sinus_Slow1;

fastSampling_sin1 := Sinus_SqSlow;  
fastSampling_sin2 := Sinus_VerySlow;
fastSampling_cosh := Cosinus_Half;  

persistent_sin1 := Sinus_SqSlow;
persistent_sin2 := Sinus_VerySlow;
persistent_cosh := Cosinus_Half;

persistent_SQL_sin1 := Sinus_SqSlow;  
persistent_SQL_sin2 := Sinus_VerySlow;
persistent_SQL_cosh := Cosinus_Half;  

(*
-----------------------------------------------------------------------------------------------------
Alarm & Conditions
-----------------------------------------------------------------------------------------------------
*)
IF( timer_1s.Q ) THEN
	limitAlmTrigger := limitAlmTrigger+1;
	IF( limitAlmTrigger > limitAlmRangeHi ) THEN
		limitAlmTrigger := limitAlmRangeLo;
	END_IF
END_IF

IF( timer_30s.Q ) THEN
	offNormAlmTrigger := NOT offNormAlmTrigger;
END_IF

IF( timer_100ms.Q ) THEN
	timer_100ms( in:=FALSE );
END_IF;

IF( timer_1s.Q ) THEN
	timer_1s( in:=FALSE );
END_IF;

IF( timer_30s.Q ) THEN
	timer_30s( in:=FALSE );
END_IF

END_PROGRAM

// ---- POUs/Programs/PRG_Static.TcPOU
PROGRAM PRG_Static
VAR
	k: INT;
	l: INT;
	m: INT;
END_VAR

	stat_scalar_BOOL	:= TRUE;
	stat_scalar_I1		:= 1;	
	stat_scalar_UI1		:= 1;	
	stat_scalar_I2 		:= 1;		
	stat_scalar_UI2		:= 1;	
	stat_scalar_I4		:= 1;	
	stat_scalar_UI4		:= 1;	
	stat_scalar_I8		:= 1;	
	stat_scalar_UI8		:= 1;	
	stat_scalar_BYTE	:= 1;	
	stat_scalar_WORD	:= 1;	
	stat_scalar_DWORD	:= 1;	
	stat_scalar_LWORD	:= 1;				
	stat_scalar_R4		:= 1.0;				
	stat_scalar_R8		:= 1.0;				
	stat_scalar_BSTR	:= 'Hello World';
	stat_scalar_WSTRING	:= "Hello World";
	stat_scalar_DT		:= DT#1972-03-29-00:00:00;
	stat_scalar_DATE 	:= DATE#1972-03-29;
	stat_scalar_TOD		:= TOD#12:00:00;	
	stat_scalar_TIME	:= T#1S;	

	GVL_structures.StructuredType1.a 			:= 42;
	GVL_structures.StructuredType1.b			:= 42;
	GVL_structures.StructuredType1.x			:= E_Enum_1.THREE;
	GVL_structures.StructuredType1.str			:= 'Hello World';

	GVL_structures.StructuredType2.c1.a			:= 42;
	GVL_structures.StructuredType2.c1.b			:= 42;
	GVL_structures.StructuredType2.c1.x			:= E_Enum_1.THREE;
	GVL_structures.StructuredType2.c1.str		:= 'Hello World';
	GVL_structures.StructuredType2.s_5			:= 'Hello';
	GVL_structures.StructuredType2.s_3			:= 'Hel';
	FOR k:= 0 TO 5 DO
		GVL_structures.StructuredType2.cArr[k].a:= 42;
		GVL_structures.StructuredType2.cArr[k].b:= 42;
		GVL_structures.StructuredType2.cArr[k].x:= E_Enum_1.THREE;
		GVL_structures.StructuredType2.cArr[k].str:= 'Hello World'; 
	END_FOR	
	GVL_structures.StructuredType2.e			:= E_Enum_1.THREE;
	FOR k:= 0 TO 100 DO
		GVL_structures.StructuredType2.iArr[k] := 42;
	END_FOR
	
	GVL_structures.StructuredType8.stComplex.a			:= 42;
	GVL_structures.StructuredType8.stComplex.b			:= 42;
	GVL_structures.StructuredType8.stComplex.x			:= E_Enum_1.THREE;
	GVL_structures.StructuredType8.stComplex.str		:= 'Hello World';
	GVL_structures.StructuredType8.strString5			:= 'Hello';
	GVL_structures.StructuredType8.strString3			:= 'Hel';
	FOR k:= 0 TO 1 DO
		GVL_structures.StructuredType8.arrComplex[k].a:= 42;
		GVL_structures.StructuredType8.arrComplex[k].b:= 42;
		GVL_structures.StructuredType8.arrComplex[k].x:= E_Enum_1.THREE;
		GVL_structures.StructuredType8.arrComplex[k].str:= 'Hello World'; 
	END_FOR	
	GVL_structures.StructuredType8.eEnum			:= E_Enum_1.THREE;
	FOR k:= 0 TO 100 DO
		GVL_structures.StructuredType8.arrDint[k] := 42;
	END_FOR	
	
	FOR k:= 0 TO ARRSIZEX DO
		stat_1dim_BOOL[k] := TRUE;
		stat_1dim_I1[k] := 1;
		stat_1dim_UI1[k] := 1;
		stat_1dim_I2[k] := 1;
		stat_1dim_UI2[k] := 1;
		stat_1dim_I4[k] := 1;
		stat_1dim_UI4[k] := 1;
		stat_1dim_I8[k] := 1;
		stat_1dim_UI8[k] := 1;
		stat_1dim_BYTE[k] := 1;
		stat_1dim_WORD[k] := 1;
		stat_1dim_DWORD[k] := 1;
		stat_1dim_LWORD[k] := 1;
		stat_1dim_R4[k] := 1.0;
		stat_1dim_R8[k] := 1.0;
		stat_1dim_BSTR[k] := 'Hello World';
		stat_1dim_WSTRING[k] := "Hello World";
		stat_1dim_DT[k] := DT#1972-03-29-00:00:00;
		stat_1dim_DATE[k] := DATE#1972-03-29;
		stat_1dim_TOD[k] := TOD#12:00:00;
		stat_1dim_TIME[k] := T#1S;
	END_FOR	

FOR l:= 0 TO ARRSIZEY DO
	FOR k:= 0 TO ARRSIZEX DO
		stat_2dim_BOOL[k,l] := TRUE;
		stat_2dim_I1[k,l] := 1;
		stat_2dim_UI1[k,l] := 1;
		stat_2dim_I2[k,l] := 1;
		stat_2dim_UI2[k,l] := 1;
		stat_2dim_I4[k,l] := 1;
		stat_2dim_UI4[k,l] := 1;
		stat_2dim_I8[k,l] := 1;
		stat_2dim_UI8[k,l] := 1;
		stat_2dim_BYTE[k,l] := 1;
		stat_2dim_WORD[k,l] := 1;
		stat_2dim_DWORD[k,l] := 1;
		stat_2dim_LWORD[k,l] := 1;
		stat_2dim_R4[k,l] := 1.0;
		stat_2dim_R8[k,l] := 1.0;
		stat_2dim_BSTR[k,l] := 'Hello World';
		stat_2dim_WSTRING[k,l] := "Hello World";
		stat_2dim_DT[k,l] := DT#1972-03-29-00:00:00;
		stat_2dim_DATE[k,l] := DATE#1972-03-29;
		stat_2dim_TOD[k,l] := TOD#12:00:00;
		stat_2dim_TIME[k,l] := T#1S;
	END_FOR
END_FOR	

FOR m:= 0 TO ARRSIZEY DO
	FOR l:= 0 TO ARRSIZEY DO
		FOR k:= 0 TO ARRSIZEX DO
			stat_3dim_BOOL[k,l,m] := TRUE;
			stat_3dim_I1[k,l,m] := 1;
			stat_3dim_UI1[k,l,m] := 1;
			stat_3dim_I2[k,l,m] := 1;
			stat_3dim_UI2[k,l,m] := 1;
			stat_3dim_I4[k,l,m] := 1;
			stat_3dim_UI4[k,l,m] := 1;
			stat_3dim_I8[k,l,m] := 1;
			stat_3dim_UI8[k,l,m] := 1;
			stat_3dim_BYTE[k,l,m] := 1;
			stat_3dim_WORD[k,l,m] := 1;
			stat_3dim_DWORD[k,l,m] := 1;
			stat_3dim_LWORD[k,l,m] := 1;
			stat_3dim_R4[k,l,m] := 1.0;
			stat_3dim_R8[k,l,m] := 1.0;
			stat_3dim_BSTR[k,l,m] := 'Hello World';
			stat_3dim_WSTRING[k,l,m] := "Hello World";
			stat_3dim_DT[k,l,m] := DT#1972-03-29-00:00:00;
			stat_3dim_DATE[k,l,m] := DATE#1972-03-29;
			stat_3dim_TOD[k,l,m] := TOD#12:00:00;
			stat_3dim_TIME[k,l,m] := T#1S;			
		END_FOR
	END_FOR
END_FOR

END_PROGRAM
